SUPER^(); // FB_BA_View
LifeSafety(); // FB_BA_EvtCategory
SafetyMsg(); // FB_BA_EvtCategory
AlarmMsg(); // FB_BA_EvtCategory
FaultMsg(); // FB_BA_EvtCategory
MaintenanceMsg01(); // FB_BA_EvtCategory
MaintenanceMsg02(); // FB_BA_EvtCategory
SystemMsg(); // FB_BA_EvtCategory
ManualOp(); // FB_BA_EvtCategory
OtherMsg(); // FB_BA_EvtCategory

METHOD FB_init : BOOL
VAR_INPUT
	bInitRetains : BOOL; // if TRUE, the retain variables are initialized (warm start / cold start)
	bInCopyCode : BOOL;  // if TRUE, the instance afterwards gets moved into the copy code (online change)
END_VAR
//===================================================================
// Ereigniskategorie - Gefahr für Leben // Event category - Danger to life
// Brandalarm, Überfall // Fire alarm, robbery
LifeSafety.iParent							:= THIS^;
LifeSafety.iLabel							:= LblCtl_EvtCategoryLifeSafty;
LifeSafety.eDPADMode						:= E_BA_DPADMode.eInclude;																						
LifeSafety.EC.nInstanceID						:= EC_ID.NC10;
LifeSafety.EC.iLabel							:= LblFun_ObjectNotificationClass;
LifeSafety.EC.sObjectName						:='{Idx=10}';
LifeSafety.EC.eAlarmMode						:= E_BA_AlarmMode.UserDefined;
LifeSafety.EC.eEventType						:= E_BA_EventType.eAlarm;
LifeSafety.EC.aPriority[1]						:= 10;
LifeSafety.EC.aPriority[2]						:= 11;
LifeSafety.EC.aPriority[3]						:= 12;
LifeSafety.EC.aAcknowledgeRequired[1]			:= TRUE;
LifeSafety.EC.aAcknowledgeRequired[2]			:= FALSE;
LifeSafety.EC.aAcknowledgeRequired[3]			:= TRUE;
//===================================================================		
// Ereigniskategorie - Gefahrenmeldung, Sicherheitsmeldung // Event category - hazard alert, safety message
// Einbruch, unberechtigter Zutritt // Burglary, unauthorised entry
SafetyMsg.iParent							:= THIS^;
SafetyMsg.iLabel							:= LblCtl_EvtCategorySaftyMessage;
SafetyMsg.eDPADMode							:= E_BA_DPADMode.eInclude;																						
SafetyMsg.EC.nInstanceID						:= EC_ID.NC20;
SafetyMsg.EC.iLabel								:= LblFun_ObjectNotificationClass;
SafetyMsg.EC.sObjectName						:='{Idx=20}';
SafetyMsg.EC.eAlarmMode							:= E_BA_AlarmMode.UserDefined;
SafetyMsg.EC.eEventType							:= E_BA_EventType.eAlarm;
SafetyMsg.EC.aPriority[1]						:= 40;
SafetyMsg.EC.aPriority[2]						:= 41;
SafetyMsg.EC.aPriority[3]						:= 42;
SafetyMsg.EC.aAcknowledgeRequired[1]			:= TRUE;
SafetyMsg.EC.aAcknowledgeRequired[2]			:= FALSE;
SafetyMsg.EC.aAcknowledgeRequired[3]			:= TRUE;
//===================================================================//
// Ereigniskategorie - Alarmeldung - Meldung signalisiert Anlagenausfall oder erfordert sofortigen Eingriff 
// Event category - Alarm message - Message signals system failure or requires immediate intervention 
// Sicherheitstemperaturbegrenzer (STB), Sicherheitsdruckbegrenzer (SDB), Übertemperatur der Warmwasserbereitung (WWB), Sicherheitsventile, Hauptpumpen, Keilriemenwächter, Frequenzumformer, Kälteanlagen, Spannungsausfall usw
// Safety temperature limiter, safety pressure limiter, excess temperature of water heating, safety valves, main pumps, V-belt monitors, frequency converters, refrigeration systems, voltage failure, etc.
AlarmMsg.iParent							:= THIS^;
AlarmMsg.iLabel								:= LblCtl_EvtCategoryAlarmMessage;
AlarmMsg.eDPADMode							:= E_BA_DPADMode.eInclude;																						
AlarmMsg.EC.nInstanceID							:= EC_ID.NC30;
AlarmMsg.EC.iLabel								:= LblFun_ObjectNotificationClass;
AlarmMsg.EC.sObjectName							:= '{Idx=30}'	;
AlarmMsg.EC.eAlarmMode							:= E_BA_AlarmMode.UserDefined;
AlarmMsg.EC.eEventType							:= E_BA_EventType.eAlarm;
AlarmMsg.EC.aPriority[1]						:= 70;
AlarmMsg.EC.aPriority[2]						:= 71;
AlarmMsg.EC.aPriority[3]						:= 72;
AlarmMsg.EC.aAcknowledgeRequired[1]				:= TRUE;
AlarmMsg.EC.aAcknowledgeRequired[2]				:= FALSE;
AlarmMsg.EC.aAcknowledgeRequired[3]				:= TRUE;

//===================================================================
// Ereigniskategorie - Störungsmeldung - Meldung weist auf einen anormalen Betriebszustand hin
// Event category - malfunction message - message indicates abnormal operating condition
// Temperaturwächter (TW), Druckwächter (DW), Temperaturüberwachung von Wärmetauscher (WT) und WWB, Motorschutz, Aufzug-Sammelstörmeldung, Netzdrücke usw.
// Temperature monitor, pressure monitor, temperature monitoring of heat exchanger and water heating, motor protection, lift collective fault signal, mains pressures, etc.
FaultMsg.iParent							:= THIS^;
FaultMsg.iLabel								:= LblCtl_EvtCategoryFaultMessage;
FaultMsg.eDPADMode							:= E_BA_DPADMode.eInclude;																						
FaultMsg.EC.nInstanceID							:= EC_ID.NC40;
FaultMsg.EC.iLabel								:= LblFun_ObjectNotificationClass;
FaultMsg.EC.sObjectName							:= '{Idx=40}'	;
FaultMsg.EC.eAlarmMode							:= E_BA_AlarmMode.UserDefined;
FaultMsg.EC.eEventType							:= E_BA_EventType.eDisturb;
FaultMsg.EC.aPriority[1]						:= 100;
FaultMsg.EC.aPriority[2]						:= 101;
FaultMsg.EC.aPriority[3]						:= 102;
FaultMsg.EC.aAcknowledgeRequired[1]				:= TRUE;
FaultMsg.EC.aAcknowledgeRequired[2]				:= FALSE;
FaultMsg.EC.aAcknowledgeRequired[3]				:= FALSE;
//===================================================================
// Ereigniskategorie - Wartungsmeldung, Hinweis auf Wartungsaktivität o.ä.
// Event category - Maintenance message Maintenance message, indication of maintenance activity or similar.
// Betriebsstunden, Behälterstand, Reparaturschalter usw.
// Operating hours, tank level, repair switch, etc.
MaintenanceMsg01.iParent					:= THIS^;
MaintenanceMsg01.iLabel						:= LblCtl_EvtCategoryMaintenanceMessage;
MaintenanceMsg01.eDPADMode					:= E_BA_DPADMode.eInclude;																						
MaintenanceMsg01.EC.nInstanceID					:= EC_ID.NC50;
MaintenanceMsg01.EC.iLabel						:= LblFun_ObjectNotificationClass;
MaintenanceMsg01.EC.sObjectName					:= '{Idx=50}'	;
MaintenanceMsg01.EC.eAlarmMode					:= E_BA_AlarmMode.UserDefined;
MaintenanceMsg01.EC.eEventType					:= E_BA_EventType.eMaintenance;
MaintenanceMsg01.EC.aPriority[1]				:= 130;
MaintenanceMsg01.EC.aPriority[2]				:= 131;
MaintenanceMsg01.EC.aPriority[3]				:= 132;
MaintenanceMsg01.EC.aAcknowledgeRequired[1]		:= TRUE;
MaintenanceMsg01.EC.aAcknowledgeRequired[2]		:= FALSE;
MaintenanceMsg01.EC.aAcknowledgeRequired[3]		:= FALSE;

// Filterende erreicht, Filter verschmutzt usw.
// Filter end reached, filter dirty, etc.
MaintenanceMsg02.iParent					:= THIS^;
MaintenanceMsg02.iLabel						:= LblCtl_EvtCategoryMaintenanceMessage;
MaintenanceMsg02.eDPADMode					:= E_BA_DPADMode.eInclude;																						
MaintenanceMsg02.EC.nInstanceID					:= EC_ID.NC51;
MaintenanceMsg02.EC.iLabel						:= LblFun_ObjectNotificationClass;
MaintenanceMsg02.EC.sObjectName					:= '{Idx=51}'	;
MaintenanceMsg02.EC.eAlarmMode					:= E_BA_AlarmMode.UserDefined;
MaintenanceMsg02.EC.eEventType					:= E_BA_EventType.eMaintenance;
MaintenanceMsg02.EC.aPriority[1]				:= 135;
MaintenanceMsg02.EC.aPriority[2]				:= 136;
MaintenanceMsg02.EC.aPriority[3]				:= 137;
MaintenanceMsg02.EC.aAcknowledgeRequired[1]		:= TRUE;
MaintenanceMsg02.EC.aAcknowledgeRequired[2]		:= FALSE;
MaintenanceMsg02.EC.aAcknowledgeRequired[3]		:= FALSE;
//===================================================================
//===================================================================
// Ereigniskategorie - Systemmeldung, Störungsmeldung aus GA-System
// Event category - System message, System message, Fault message from building automation system
// Gerätestörung, Batteriemeldung, Kommunikationsunterbrechung usw.
// Unit malfunction, battery message, communication interruption, etc.
SystemMsg.iParent							:= THIS^;
SystemMsg.iLabel							:= LblCtl_EvtCategorySystem;
SystemMsg.eDPADMode							:= E_BA_DPADMode.eInclude;																						
SystemMsg.EC.nInstanceID						:= EC_ID.NC60;
SystemMsg.EC.iLabel								:= LblFun_ObjectNotificationClass;
SystemMsg.EC.sObjectName						:='{Idx=60}';
SystemMsg.EC.eAlarmMode							:= E_BA_AlarmMode.UserDefined;
SystemMsg.EC.eEventType							:= E_BA_EventType.eNotification;
SystemMsg.EC.aPriority[1]						:= 180;
SystemMsg.EC.aPriority[2]						:= 181;
SystemMsg.EC.aPriority[3]						:= 182;
SystemMsg.EC.aAcknowledgeRequired[1]			:= FALSE;
SystemMsg.EC.aAcknowledgeRequired[2]			:= FALSE;
SystemMsg.EC.aAcknowledgeRequired[3]			:= FALSE;
//===================================================================//
//	Ereigniskategorie - Manual operation, Handeingriff
ManualOp.iParent							:= THIS^;
ManualOp.iLabel								:= LblCtl_EvtCategoryManualOperation;
ManualOp.eDPADMode							:= E_BA_DPADMode.eInclude;																						
ManualOp.EC.nInstanceID							:= EC_ID.NC70;
ManualOp.EC.iLabel								:= LblFun_ObjectNotificationClass;
ManualOp.EC.sObjectName							:='{Idx=70}';
ManualOp.EC.eAlarmMode							:= E_BA_AlarmMode.UserDefined;
ManualOp.EC.eEventType							:= E_BA_EventType.eOther;
ManualOp.EC.aPriority[1]						:= 220;
ManualOp.EC.aPriority[2]						:= 220;
ManualOp.EC.aPriority[3]						:= 220;
ManualOp.EC.aAcknowledgeRequired[1]				:= FALSE;
ManualOp.EC.aAcknowledgeRequired[2]				:= FALSE;
ManualOp.EC.aAcknowledgeRequired[3]				:= FALSE;
//===================================================================//
// Ereigniskategorie - Freibleibend, Sonstige Meldungen
// Event category - Other message, Not binding, Other messages
// Betriebszustandswechsel, Betriebsarten, Trendspeicher voll usw.
// Operating status change, operating modes, trend memory full, etc.
OtherMsg.iParent							:= THIS^;
OtherMsg.iLabel								:= LblCtl_EvtCategoryOther;
OtherMsg.eDPADMode							:= E_BA_DPADMode.eInclude;																						
OtherMsg.EC.nInstanceID							:= EC_ID.NC80;
OtherMsg.EC.iLabel								:= LblFun_ObjectNotificationClass;
OtherMsg.EC.sObjectName							:='{Idx=80}';
OtherMsg.EC.eAlarmMode							:= E_BA_AlarmMode.UserDefined;
OtherMsg.EC.eEventType							:= E_BA_EventType.eOther;
OtherMsg.EC.aPriority[1]						:= 230;
OtherMsg.EC.aPriority[2]						:= 231;
OtherMsg.EC.aPriority[3]						:= 232;
OtherMsg.EC.aAcknowledgeRequired[1]				:= FALSE;
OtherMsg.EC.aAcknowledgeRequired[2]				:= FALSE;
OtherMsg.EC.aAcknowledgeRequired[3]				:= FALSE;
END_METHOD

END_FUNCTION_BLOCK

// ---- Templates/POUs/Trade/BuildingAutomation/Communication/FB_BA_AdsComClient.TcPOU
FUNCTION_BLOCK FB_BA_AdsComClient EXTENDS FB_BA_VIEW
VAR_INPUT
END_VAR
VAR_OUTPUT
END_VAR
VAR_INPUT CONSTANT
	WeatherStation					: FB_BA_RawSubscriber;
	WeatherStationError				: FB_BA_BV;											

	GeneralSettings					: FB_BA_RawSubscriber;												
	GeneralSettingsError			: FB_BA_BV;			
END_VAR
VAR
END_VAR

// Error-notification
WeatherStationError(bEnPgm := TRUE, bValPgm := WeatherStation.bError); // FB_BA_BV
GeneralSettingsError(bEnPgm := TRUE, bValPgm := GeneralSettings.bError); // FB_BA_BV
// variable, on which the error-notification is written
Site.bWeatherStation_Error := WeatherStationError.bEvent;
// variable, on which the subscribed data is written
// because this variable is an announcement for the suscriber,
// where to write the data, it is declared as an input
// error-delay: see FB_Init
WeatherStation(xData := Site.stWeatherStation); // FB_BA_RawSubscriber
Site.bGeneralSettings_Error := GeneralSettingsError.bEvent;
GeneralSettings(xData := Site.stGeneralSettings); // FB_BA_RawSubscriber
SUPER^(); // FB_BA_VIEW

METHOD FB_init : BOOL
VAR_INPUT
	bInitRetains : BOOL; // if TRUE, the retain variables are initialized (warm start / cold start)
	bInCopyCode : BOOL;  // if TRUE, the instance afterwards gets moved into the copy code (online change)
END_VAR
WeatherStation.Subject							:= Site.WeatherStation_Subject;		// instance-name of the publisher in the source
WeatherStation.sTarget							:= Site.WeatherStation_NetId;		// AMS-Net-Id of the publishing controller
WeatherStation.tReadInterval					:= T#5S;							// subscribe-interval
WeatherStation.tReadTolerance					:= T#60S;							// delay time, until an erroneous communication will be displayed at the error-output of the subscriber

WeatherStationError.iParent						:= THIS^;
WeatherStationError.iLabel						:= LblAgg_WeatherStationComm;
WeatherStationError.sActiveText 				:= txtEvent_Triggered;
WeatherStationError.sInactiveText 				:= txtEvent_Normal;
WeatherStationError.bEnManualRm					:= FALSE;	//	Priority  8	
WeatherStationError.bValManualRm				:= FALSE;	//	Priority  8
WeatherStationError.nEventClassID				:= EC_ID.NC30;
WeatherStationError.stTimeDelay.nToNormal		:= 0;
WeatherStationError.stTimeDelay.nToAbnormal		:= 0;
WeatherStationError.bAlarmValue					:= TRUE;
WeatherStationError.aEventTransitionText[1]		:= txtEvent_Disturb;
WeatherStationError.aEventTransitionText[2]		:= txtEvent_None;
WeatherStationError.aEventTransitionText[3]		:= txtEvent_Normal;
WeatherStationError.bEventDetectionEnable		:= TRUE;
WeatherStationError.eEnPlantLock				:= E_BA_LockPriority.eNoLock;

GeneralSettings.Subject							:= Site.GeneralSettings_Subject;	// instance-name of the publisher in the source
GeneralSettings.sTarget							:= Site.GeneralSettings_NetId;		// AMS-Net-Id of the publishing controller
GeneralSettings.tReadInterval					:= T#5S;							// subscribe-interval
GeneralSettings.tReadTolerance					:= T#60S;							// delay time, until an erroneous communication will be displayed at the error-output of the subscriber

GeneralSettingsError.iParent					:= THIS^;
GeneralSettingsError.iLabel						:= LblAgg_GeneralSettingsCom;
//GeneralSettingsError.sObjectName				:= F_BA_CONCAT06(s01:= Seperator.sAgg_ObjName, s02:= Agg_GeneralSettingsCom_ObjName, s03:= '02', s04:= Seperator.sFun_ObjName, s05:= Fun_Fault_ObjName, s06:= '01');  
//GeneralSettingsError.sDescription				:= F_BA_CONCAT06(s01:= Seperator.sAgg_Descr, s02:= Agg_GeneralSettingsCom_Descr, s03:= '', s04:= Seperator.sFun_Descr, s05:= Fun_Fault_Descr, s06:= ''); 	
GeneralSettingsError.sActiveText 				:= txtEvent_Triggered;
GeneralSettingsError.sInactiveText 				:= txtEvent_Normal;
GeneralSettingsError.bEnManualRm				:= FALSE;	//	Priority  8	
GeneralSettingsError.bValManualRm				:= FALSE;	//	Priority  8
GeneralSettingsError.nEventClassID				:= EC_ID.NC30;
GeneralSettingsError.stTimeDelay.nToNormal		:= 0;
GeneralSettingsError.stTimeDelay.nToAbnormal	:= 0;
GeneralSettingsError.bAlarmValue				:= TRUE;
GeneralSettingsError.aEventTransitionText[1]	:= txtEvent_Disturb;
GeneralSettingsError.aEventTransitionText[2]	:= txtEvent_None;
GeneralSettingsError.aEventTransitionText[3]	:= txtEvent_Normal;
GeneralSettingsError.bEventDetectionEnable		:= TRUE;
GeneralSettingsError.eEnPlantLock				:= E_BA_LockPriority.eNoLock;
END_METHOD

END_FUNCTION_BLOCK

// ---- Templates/POUs/Trade/HeatingSystem/General/FB_BA_HtgLmt.TcPOU
{region '#Template'}
	{attribute 'Version' := '5.0.0.0'}
	{attribute 'Tags' := '"LCID": "1031", "Text": "H, General, HtgCir, Operating mode"'}
	{attribute 'Tags' := '"LCID": "1033", "Text": "H, General, HtgCir, Operating mode"'}
	{attribute 'Using' := '"Type": "Template", "URI": "BA2_Param"'}
	{attribute 'Description' := '"LCID": "1031", "Text": "Heizgrenzwert"'}
	{attribute 'Description' := '"LCID": "1033", "Text": "Heating limit"'}
{endregion}
FUNCTION_BLOCK FB_BA_HtgLmt EXTENDS FB_BA_View
VAR_INPUT
	fIn						: REAL;
END_VAR
VAR_OUTPUT
	bQ						: BOOL;
END_VAR
VAR_INPUT CONSTANT
	Sp						: FB_BA_AV_Op;	
	Q						: FB_BA_BV_Op;		
END_VAR	
VAR
	Swi2P					: FB_BA_Swi2P;
END_VAR
VAR // added by the converter: edge detectors and wires of the graphical bodies
    _w1 : ANY;
END_VAR

SUPER^(); // FB_BA_View
Sp(); // FB_BA_AV_Op
_w1 := LIMIT(10, Sp.fPresentValue, 32);
Swi2P(bEn := TRUE, fIn := fIn, fOn := _w1, fOff := _w1 + 0.5); // FB_BA_Swi2P
Q(bValuePgm := Swi2P.bQ); // FB_BA_BV_Op
bQ := Q.bPresentValue;

METHOD FB_init : BOOL
VAR_INPUT
	bInitRetains : BOOL; // if TRUE, the retain variables are initialized (warm start / cold start)
	bInCopyCode : BOOL;  // if TRUE, the instance afterwards gets moved into the copy code (online change)
END_VAR
Sp.iParent			:= THIS^;
Sp.iLabel			:= LblFun_Setpoint; 
Sp.eUnit			:= E_BA_Unit.eTemperature_DegreesCelsius;  
Sp.fValueRm			:= 16.0;
Sp.fCOVIncrement	:= BA2_Param.fDefCOVIncrement;							

Q.iParent			:= THIS^;
Q.iLabel			:= LblFun_OperationalMessage; 
Q.sActiveText		:= txtEvent_On;
Q.sInactiveText		:= txtEvent_Off;
Q.bValueRm			:= FALSE;								
Q.eToggleMode 		:= E_BA_ToggleMode.eSwitch;
END_METHOD

END_FUNCTION_BLOCK

// ---- Templates/POUs/Trade/HeatingSystem/Setpoint/FB_BA_H_HtgCir_Sp.TcPOU
{region '#Template'}
	{attribute 'Version' := '5.0.0.0'}
	{attribute 'Tags' := '"LCID": "1031", "Text": "H, Heating circuit, HtgCir, Setpoint"'}
	{attribute 'Tags' := '"LCID": "1033", "Text": "H, Heating circuit, HtgCir, Setpoint"'}
	{attribute 'Using' := '"Type": "Template", "URI": "BA2_Param"'}
	{attribute 'Using' := '"Type": "Template", "URI": "E_BA_EnergyLvl"'}		 
	{attribute 'Description' := '"LCID": "1031", "Text": "Sollwert Heizkreis"'}
	{attribute 'Description' := '"LCID": "1033", "Text": "Setpoint heating circuit"'}
{endregion}
FUNCTION_BLOCK FB_BA_H_HtgCir_Sp EXTENDS FB_BA_View
VAR_INPUT
	eOpMod					: E_BA_EnergyLvl;
	fSpFrstProtec			: REAL;
	fTWthDamp				: REAL;
END_VAR
VAR_OUTPUT
	fSpFlWT							: REAL;
END_VAR
VAR_INPUT CONSTANT
	NgtOffs					: FB_BA_AV_Op;	
	SpFlWT					: FB_BA_AV_Op;		
	HtgCrv					: FB_BA_Scale_04; 
END_VAR
VAR
	PrioSwi					: FB_BA_MMUX_R04;
END_VAR

// note: 1 stored wires end on pins the file does not list and are not shown
SUPER^(); // FB_BA_View
NgtOffs(); // FB_BA_AV_Op
HtgCrv(fX := fTWthDamp); // FB_BA_Scale_04
PrioSwi(
    bEn := TRUE,
    nSel := eOpMod,
    nEn01 := E_BA_EnergyLvl.eComfort,
    fVal01 := HtgCrv.fY,
    nEn02 := E_BA_EnergyLvl.eEconomy,
    fVal02 := HtgCrv.fY - ABS(NgtOffs.fPresentValue),
    nEn03 := E_BA_EnergyLvl.eProtection,
    fVal03 := fSpFrstProtec); // FB_BA_MMUX_R04
SpFlWT(fValuePgm := PrioSwi.fVal); // FB_BA_AV_Op
fSpFlWT := SpFlWT.fPresentValue;

METHOD FB_init : BOOL
VAR_INPUT
	bInitRetains : BOOL; // if TRUE, the retain variables are initialized (warm start / cold start)
	bInCopyCode : BOOL;  // if TRUE, the instance afterwards gets moved into the copy code (online change)
END_VAR
NgtOffs.iParent				:= THIS^;
NgtOffs.iLabel				:= LblCtl_OffsetNightSetpoint; 
NgtOffs.eUnit				:= E_BA_Unit.eTemperature_DegreesCelsius;  
NgtOffs.fValueRm			:= 8.0;
NgtOffs.fCOVIncrement		:= BA2_Param.fDefCOVIncrement;							

SpFlWT.iParent				:= THIS^;
SpFlWT.iLabel				:= LblFun_Setpoint; 
SpFlWT.eUnit				:= E_BA_Unit.eTemperature_DegreesCelsius;  
SpFlWT.fCOVIncrement		:= BA2_Param.fDefCOVIncrement;							

HtgCrv.iParent				:= THIS^;										
HtgCrv.iLabel				:= LblCtl_HeatingCurve; 
HtgCrv.eDPADMode			:= E_BA_DPADMode.eIncludeDescription; 
HtgCrv.X1.fValueRm			:= 15.0;
HtgCrv.X2.fValueRm			:= 0.0;
HtgCrv.X3.fValueRm			:= -10.0;
HtgCrv.X4.fValueRm			:= -20.0;
HtgCrv.Y1.fValueRm			:= 25.0;
HtgCrv.Y2.fValueRm			:= 40.0;
HtgCrv.Y3.fValueRm			:= 55.0;
HtgCrv.Y4.fValueRm			:= 65.0;
HtgCrv.YMin.fValueRm		:= 5.0;
HtgCrv.YMax.fValueRm		:= 80.0;
END_METHOD

END_FUNCTION_BLOCK

// ---- Templates/POUs/Universal/Control/Scale/FB_BA_Scale_04.TcPOU
{region '#Template'}
	{attribute 'Version' := '5.0.0.0'}
	{attribute 'Tags' := '"LCID": "1031", "Text": "Universal, Control, Scaling"'}
	{attribute 'Tags' := '"LCID": "1033", "Text": "Universal, Control, Scaling"'}
	{attribute 'Using' := '"Type": "Template", "URI": "BA2_Param"'}
	{attribute 'Description' := '"LCID": "1031", "Text": "Skalierung"'}
	{attribute 'Description' := '"LCID": "1033", "Text": "Scaling"'}
{endregion}
FUNCTION_BLOCK FB_BA_Scale_04 EXTENDS FB_BA_View
VAR_INPUT
	fX			: REAL;
END_VAR
VAR_OUTPUT
	fY			: REAL;
END_VAR
VAR_INPUT CONSTANT
	X1			: FB_BA_AV_Op;	
	X2			: FB_BA_AV_Op;	
	X3			: FB_BA_AV_Op;	
	X4			: FB_BA_AV_Op;	
	Y1			: FB_BA_AV_Op;	
	Y2			: FB_BA_AV_Op;
	Y3			: FB_BA_AV_Op;
	Y4			: FB_BA_AV_Op;
	YMin		: FB_BA_AV_Op;			
	YMax		: FB_BA_AV_Op;			
	Y			: FB_BA_AV_Op;		
END_VAR
VAR		
	Scale		: FB_BA_Chrct04;
END_VAR

SUPER^(); // FB_BA_View
X1(); // FB_BA_AV_Op
X2(); // FB_BA_AV_Op
X3(); // FB_BA_AV_Op
X4(); // FB_BA_AV_Op
Y1(); // FB_BA_AV_Op
Y2(); // FB_BA_AV_Op
Y3(); // FB_BA_AV_Op
Y4(); // FB_BA_AV_Op
Ymin(); // FB_BA_AV_Op
YMax(); // FB_BA_AV_Op
Scale(
    fX := fX,
    fX01 := X1.fPresentValue,
    fX02 := X2.fPresentValue,
    fX03 := X3.fPresentValue,
    fX04 := X4.fPresentValue,
    fY01 := Y1.fPresentValue,
    fY02 := Y2.fPresentValue,
    fY03 := Y3.fPresentValue,
    fY04 := Y4.fPresentValue,
    fYMin := Ymin.fPresentValue,
    fYMax := YMax.fPresentValue); // FB_BA_Chrct04
Y(fValuePgm := Scale.fCalcVal); // FB_BA_AV_Op
fY := Y.fPresentValue;

METHOD FB_init : BOOL
VAR_INPUT
	bInitRetains : BOOL; // if TRUE, the retain variables are initialized (warm start / cold start)
	bInCopyCode : BOOL;  // if TRUE, the instance afterwards gets moved into the copy code (online change)
END_VAR
X1.iParent			:= THIS^;
X1.iLabel		:= LblCtl_X01;  							 	 
X1.eUnit			:= E_BA_Unit.eTemperature_DegreesCelsius;						 	 
X1.fValueRm			:= 15.0;
X1.fCOVIncrement	:= BA2_Param.fDefCOVIncrement;		

X2.iParent			:= THIS^;
X2.iLabel		:= LblCtl_X02;  								 	 
X2.eUnit			:= E_BA_Unit.eTemperature_DegreesCelsius;						 	 
X2.fValueRm			:= 0.0;
X2.fCOVIncrement	:= BA2_Param.fDefCOVIncrement;		

X3.iParent			:= THIS^;
X3.iLabel		:= LblCtl_X03;  								 	 
X3.eUnit			:= E_BA_Unit.eTemperature_DegreesCelsius;						 	 
X3.fValueRm			:= -20.0;
X3.fCOVIncrement	:= BA2_Param.fDefCOVIncrement;			

X4.iParent			:= THIS^;
X4.iLabel		:= LblCtl_X04;  									 	 
X4.eUnit			:= E_BA_Unit.eTemperature_DegreesCelsius;						 	 
X4.fValueRm			:= -20.0;
X4.fCOVIncrement	:= BA2_Param.fDefCOVIncrement;		

Y1.iParent			:= THIS^;
Y1.iLabel		:= LblCtl_Y01;  			 	 
Y1.eUnit			:= E_BA_Unit.eTemperature_DegreesCelsius;						 	 
Y1.fValueRm			:= 25.0;
Y1.fCOVIncrement	:= BA2_Param.fDefCOVIncrement;		

Y2.iParent			:= THIS^;
Y2.iLabel		:= LblCtl_Y02;  							 	 
Y2.eUnit			:= E_BA_Unit.eTemperature_DegreesCelsius;						 	 
Y2.fValueRm			:= 40.0;
Y2.fCOVIncrement	:= BA2_Param.fDefCOVIncrement;		

Y3.iParent			:= THIS^;
Y3.iLabel			:= LblCtl_Y03;  							 	 
Y3.eUnit			:= E_BA_Unit.eTemperature_DegreesCelsius;						 	 
Y3.fValueRm			:= 60.0;
Y3.fCOVIncrement	:= BA2_Param.fDefCOVIncrement;		


Y4.iParent			:= THIS^;
Y4.iLabel			:= LblCtl_Y04;  									 	 
Y4.eUnit			:= E_BA_Unit.eTemperature_DegreesCelsius;						 	 
Y4.fValueRm			:= 65.0;
Y4.fCOVIncrement	:= BA2_Param.fDefCOVIncrement;		

YMin.iParent		:= THIS^;
YMin.iLabel			:= LblFun_MinimumValue;										 	 
YMin.eUnit			:= E_BA_Unit.eTemperature_DegreesCelsius;						 	 
YMin.fValueRm		:= 5.0;
YMin.fCOVIncrement	:= BA2_Param.fDefCOVIncrement;		

YMax.iParent		:= THIS^;
YMax.iLabel			:= LblFun_MaximumValue;							 	 
YMax.eUnit			:= E_BA_Unit.eTemperature_DegreesCelsius;						 	 
YMax.fValueRm		:= 80.0;
YMax.fCOVIncrement	:= BA2_Param.fDefCOVIncrement;		

Y.iParent			:= THIS^;
Y.iLabel			:= LblFun_SetpointCalculated;										 	 
Y.eUnit				:= E_BA_Unit.eTemperature_DegreesCelsius;	
Y.fCOVIncrement		:= BA2_Param.fDefCOVIncrement;
END_METHOD

END_FUNCTION_BLOCK

// ---- Templates/POUs/Universal/Aggregat/Analog/FB_BA_ActuatorAV.TcPOU
{region '#Template'}
	{attribute 'Version' := '5.0.0.0'}
	{attribute 'Tags' := '"LCID": "1031", "Text": "Universal, Analog, Aggregate"'}
	{attribute 'Tags' := '"LCID": "1033", "Text": "Universal, Analog, Aggregate"'}
	{attribute 'Using' := '"Type": "Template", "URI": "EC_ID"'}
	{attribute 'Using' := '"Type": "Template", "URI": "BA2_Param"'}
	{attribute 'Description' := '"LCID": "1031", "Text": "AV"'}
	{attribute 'Description' := '"LCID": "1033", "Text": "AV"'}
{endregion}
FUNCTION_BLOCK FB_BA_ActuatorAV EXTENDS FB_BA_View
VAR_INPUT
	stCmd					: ST_BA_Analog;	
END_VAR
VAR_OUTPUT
	fPresentValue		: REAL;
	bDst				: BOOL;
	eActivePrio			: E_BA_Priority;	
END_VAR
VAR_INPUT CONSTANT
	Val					: FB_BA_AV;		
	PlantLock			: FB_BA_PlantLock;	
END_VAR
VAR
	bPrioSfty				: BOOL;
	bPrioCrit				: BOOL;	
END_VAR

SUPER^(); // FB_BA_View
PlantLock(); // FB_BA_PlantLock
bPrioSfty := PlantLock.bPrioHigh OR PlantLock.bPrioLocalHigh;
bPrioCrit := PlantLock.bPrioMedium OR PlantLock.bPrioLocalMedium;
bDst := bPrioSfty OR bPrioCrit;
Val(
    bEnSfty := stCmd.bEnSfty OR bPrioSfty,
    fValSfty := SEL(bPrioSfty, stCmd.fValSfty, 0),
    bEnCrit := stCmd.bEnCrit OR bPrioCrit,
    fValCrit := SEL(bPrioCrit, stCmd.fValCrit, 0),
    bEnPgm := stCmd.bEnPgm,
    fValPgm := stCmd.fValPgm); // FB_BA_AV
fPresentValue := Val.fPresentValue;
eActivePrio := Val.eActivePrio;

METHOD FB_init : BOOL
VAR_INPUT
	bInitRetains : BOOL; // if TRUE, the retain variables are initialized (warm start / cold start)
	bInCopyCode : BOOL;  // if TRUE, the instance afterwards gets moved into the copy code (online change)
END_VAR
PlantLock.Parent				:= THIS^;		

Val.iParent						:= THIS^;
Val.iLabel						:= LblFun_ControlSignal;  
Val.eUnit						:= E_BA_Unit.eOther_Percent;
Val.fCOVIncrement				:= BA2_Param.fDefCOVIncrement;
Val.bEnManualRm					:= FALSE;	//	Priority  8	
Val.fValManualRm				:= 0.0;		//	Priority  8
Val.fDefaultValue				:= 0.0;	
Val.nEventClassID				:= EC_ID.NC80;
Val.stTimeDelay.nToNormal		:= BA2_Param.nDefTimeDelay_ToNormal;
Val.stTimeDelay.nToAbnormal		:= BA2_Param.nDefTimeDelay_ToAbnormal;
Val.stHighLimit.bEnable			:= FALSE;
Val.stHighLimit.fValue			:= 0.0;		
Val.stLowLimit.bEnable			:= FALSE;
Val.stLowLimit.fValue			:= 0.0;
Val.fLimitDeadband 				:= BA2_Param.fDefLimitDeadband;
Val.bAcknowledgeRm				:= FALSE;	
Val.aEventTransitionText[1]		:= txtEvent_Disturb;
Val.aEventTransitionText[2]		:= txtEvent_None;
Val.aEventTransitionText[3]		:= txtEvent_Normal;
Val.bEventDetectionEnable		:= FALSE;
Val.eEnPlantLock				:= E_BA_LockPriority.eNoLock;
END_METHOD

END_FUNCTION_BLOCK

// ---- Templates/POUs/Universal/Aggregat/Modulation/FB_BA_ActuatorMdlt.TcPOU
{region '#Template'}
	{attribute 'Version' := '5.0.0.0'}
	{attribute 'Tags' := '"LCID": "1031", "Text": "Universal, Analog, Aggregate"'}
	{attribute 'Tags' := '"LCID": "1033", "Text": "Universal, Analog, Aggregate"'}
	{attribute 'Using' := '"Type": "Template", "URI": "EC_ID"'}
	{attribute 'Using' := '"Type": "Template", "URI": "BA2_Param"'}
	{attribute 'Description' := '"LCID": "1031", "Text": "Aktor analog"'}
	{attribute 'Description' := '"LCID": "1033", "Text": "Actuator analog"'}
{endregion}
FUNCTION_BLOCK FB_BA_ActuatorMdlt EXTENDS FB_BA_View
VAR_INPUT
	stCmd					: ST_BA_Mdlt;	
	fValPgm					: REAL;
END_VAR
VAR_OUTPUT
	fMdlt					: REAL;
	bDst					: BOOL;
	eActivePrio				: E_BA_Priority;
END_VAR
VAR_INPUT CONSTANT PERSISTENT
	{attribute 'parameterCategory' := 'Behaviour'}
	fMinModulation 				: REAL := 20;
	{attribute 'parameterCategory' := 'Behaviour'}
	fMaxModulation 				: REAL := 100;
END_VAR
VAR_INPUT CONSTANT
	Mdlt					: FB_BA_AO_Raw;
	PlantLock				: FB_BA_PlantLock;	
END_VAR
VAR
	bPrioSfty					: BOOL;
	bPrioCrit					: BOOL;	
	
	PrioSwiVal					: FB_BA_PrioSwi_UDI04;	
	MuxMdlt						: FB_BA_MMUX_R04;
END_VAR

SUPER^(); // FB_BA_View
PlantLock(); // FB_BA_PlantLock
bPrioSfty := PlantLock.bPrioHigh OR PlantLock.bPrioLocalHigh;
bPrioCrit := PlantLock.bPrioMedium OR PlantLock.bPrioLocalMedium;
bDst := bPrioSfty OR bPrioCrit;
PrioSwiVal(
    bEn01 := stCmd.bEnSfty,
    nVal01 := stCmd.eValSfty,
    bEn02 := stCmd.bEnCrit,
    nVal02 := stCmd.eValCrit,
    bEn03 := stCmd.bEnPgm,
    nVal03 := stCmd.eValPgm); // FB_BA_PrioSwi_UDI04
MuxMdlt(
    bEn := TRUE,
    nSel := PrioSwiVal.nVal,
    nEn01 := E_BA_Mdlt.eOff,
    fVal01 := 0,
    nEn02 := E_BA_Mdlt.eOn,
    fVal02 := fValPgm,
    nEn03 := E_BA_Mdlt.eMin,
    fVal03 := fMinModulation,
    nEn04 := E_BA_Mdlt.eMax,
    fVal04 := fMaxModulation); // FB_BA_MMUX_R04
Mdlt(
    bEnSfty := stCmd.bEnSfty,
    fValSfty := SEL(bPrioSfty, MuxMdlt.fVal, 0),
    bEnCrit := stCmd.bEnCrit,
    fValCrit := SEL(bPrioCrit, MuxMdlt.fVal, 0),
    bEnPgm := stCmd.bEnPgm,
    fValPgm := MuxMdlt.fVal); // FB_BA_AO_Raw
fMdlt := Mdlt.fPresentValue;
eActivePrio := Mdlt.eActivePrio;

METHOD FB_init : BOOL
VAR_INPUT
	bInitRetains : BOOL; // if TRUE, the retain variables are initialized (warm start / cold start)
	bInCopyCode : BOOL;  // if TRUE, the instance afterwards gets moved into the copy code (online change)
END_VAR
PlantLock.Parent				:= THIS^;		

Mdlt.iParent					:= THIS^;
Mdlt.iLabel						:= LblFun_ControlSignal;
Mdlt.eUnit						:= E_BA_Unit.eOther_Percent;
Mdlt.fResolution 				:= 0.003051851;
Mdlt.fScaleOffset 				:= 0;
Mdlt.fCOVIncrement				:= BA2_Param.fDefCOVIncrement;
Mdlt.bEnManualRm				:= FALSE;	//	Priority  8	
Mdlt.fValManualRm				:= 0.0;		//	Priority  8
Mdlt.nEventClassID				:= EC_ID.NC80;
Mdlt.stTimeDelay.nToNormal		:= BA2_Param.nDefTimeDelay_ToNormal;
Mdlt.stTimeDelay.nToAbnormal	:= BA2_Param.nDefTimeDelay_ToAbnormal;
Mdlt.stHighLimit.bEnable		:= FALSE;
Mdlt.stHighLimit.fValue			:= 0.0;		
Mdlt.stLowLimit.bEnable			:= FALSE;
Mdlt.stLowLimit.fValue			:= 0.0;
Mdlt.fLimitDeadband 			:= BA2_Param.fDefLimitDeadband;
Mdlt.aEventTransitionText[1]	:= txtEvent_Disturb;
Mdlt.aEventTransitionText[2]	:= txtEvent_None;
Mdlt.aEventTransitionText[3]	:= txtEvent_Normal;
Mdlt.bEventDetectionEnable		:= FALSE;
Mdlt.eEnPlantLock				:= E_BA_LockPriority.eNoLock;
END_METHOD

END_FUNCTION_BLOCK

// ---- Templates/POUs/Universal/Aggregat/Multistate/FB_BA_ActuatorMultistate.TcPOU
{region '#Template'}
	{attribute 'Version' := '5.0.0.0'}
	{attribute 'Tags' := '"LCID": "1031", "Text": "Universal, Multistate, Aggregate"'}
	{attribute 'Tags' := '"LCID": "1033", "Text": "Universal, Multistate, Aggregate"'}
	{attribute 'Using' := '"Type": "Template", "URI": "EC_ID"'}
	{attribute 'Using' := '"Type": "Template", "URI": "BA2_Param"'}
	{attribute 'Description' := '"LCID": "1031", "Text": "Aktor multistate"'}
	{attribute 'Description' := '"LCID": "1033", "Text": "Actuator multistate"'}
{endregion}			 
FUNCTION_BLOCK FB_BA_ActuatorMultistate EXTENDS FB_BA_View
VAR_INPUT
	stCmd					: ST_BA_Multistate;	
END_VAR
VAR_OUTPUT
	nCmd					: UDINT;
	bDst					: BOOL;
	eActivePrio				: E_BA_Priority;
END_VAR
VAR_INPUT CONSTANT	
	Cmd						: FB_BA_MO_Raw;	
	PlantLock				: FB_BA_PlantLock;	
END_VAR
VAR
	bPrioSfty				: BOOL;
	bPrioCrit				: BOOL;	
END_VAR
VAR // added by the converter: edge detectors and wires of the graphical bodies
    _w1 : ANY;
END_VAR

SUPER^(); // FB_BA_View
PlantLock(); // FB_BA_PlantLock
bPrioSfty := PlantLock.bPrioHigh OR PlantLock.bPrioLocalHigh;
bPrioCrit := PlantLock.bPrioMedium OR PlantLock.bPrioLocalMedium;
bDst := bPrioSfty OR bPrioCrit;
Cmd(
    bEnSfty := stCmd.bEnSfty OR bPrioSfty,
    nValSfty := SEL(bPrioSfty, stCmd.nValSfty, 1),
    bEnCrit := stCmd.bEnCrit OR bPrioCrit,
    nValCrit := _w1,
    bEnPgm := stCmd.bEnPgm,
    nValPgm := stCmd.nValPgm); // FB_BA_MO_Raw
_w1 := SEL(bPrioCrit, stCmd.nValCrit, 1);
nCmd := Cmd.nPresentValue;
eActivePrio := Cmd.eActivePrio;

METHOD FB_init : BOOL
VAR_INPUT
	bInitRetains : BOOL; // if TRUE, the retain variables are initialized (warm start / cold start)
	bInCopyCode : BOOL;  // if TRUE, the instance afterwards gets moved into the copy code (online change)
END_VAR
PlantLock.Parent				:= THIS^;	

Cmd.iParent						:= THIS^;
Cmd.iLabel						:= LblFun_SwitchingCommand;
Cmd.aStateText[1]				:= txtEvent_Stop;
Cmd.aStateText[2]				:= txtEvent_Open;
Cmd.aStateText[3]				:= txtEvent_Close;
Cmd.bEnManualRm					:= FALSE;	//	Priority  8	
Cmd.nValManualRm				:= 1;		//	Priority  8
Cmd.nDefaultValue				:= 1;	
Cmd.nEventClassID				:= EC_ID.NC80;
Cmd.stTimeDelay.nToNormal		:= BA2_Param.nDefTimeDelay_ToNormal;
Cmd.stTimeDelay.nToAbnormal		:= BA2_Param.nDefTimeDelay_ToAbnormal;
Cmd.aEventTransitionText[1]		:= txtEvent_Disturb;
Cmd.aEventTransitionText[2]		:= txtEvent_None;
Cmd.aEventTransitionText[3]		:= txtEvent_Normal;
Cmd.bEventDetectionEnable		:= FALSE;
Cmd.eEnPlantLock				:= E_BA_LockPriority.eNoLock;
Cmd.eMappingMode				:= E_BA_ByteMappingMode.eBinaryDecimal;
Cmd.eFeedbackMappingMode		:= E_BA_ByteMappingMode.eBinaryDecimal;
END_METHOD

END_FUNCTION_BLOCK

// ---- Templates/POUs/Universal/Control/Monitoring/FB_BA_FdbBinary.TcPOU
{region '#Template'}
	{attribute 'Version' := '5.0.0.0'}
	{attribute 'Tags' := '"LCID": "1031", "Text": "Universal, Control, Monitoring"'}
	{attribute 'Tags' := '"LCID": "1033", "Text": "Universal, Control, Monitoring"'}
	{attribute 'Using' := '"Type": "Template", "URI": "EC_ID"'}
	{attribute 'Using' := '"Type": "Template", "URI": "BA2_Param"'}
	{attribute 'Description' := '"LCID": "1031", "Text": "Überwachung von Signalen"'}
	{attribute 'Description' := '"LCID": "1033", "Text": "Monitoring signals"'}
{endregion}
FUNCTION_BLOCK FB_BA_FdbBinary EXTENDS FB_BA_View
VAR_INPUT
	bEn						: BOOL;	
	bCommand				: BOOL;	
	bFeedback				: BOOL;		
END_VAR
VAR_OUTPUT
	bDst					: BOOL;
END_VAR
VAR_INPUT CONSTANT
	DelayFeedback			: FB_BA_AV_Op;
	Dst						: FB_BA_BV;			
END_VAR
VAR_INPUT CONSTANT PERSISTENT
	{attribute 'parameterUnit':= 's'}
	nInterruptionDelay : UDINT := 1;
END_VAR
VAR
	FdbCtrl					: FB_BA_FdbCtrlBinary;		
END_VAR

SUPER^(); // FB_BA_View
DelayFeedback(); // FB_BA_AV_Op
FdbCtrl(
    bEn := bEn,
    bActuator := bCommand,
    bSwitch := bFeedback,
    nFdbDelay := TO_UDINT(DelayFeedback.fPresentValue),
    nInterruptionDelay := nInterruptionDelay); // FB_BA_FdbCtrlBinary
Dst(bEnPgm := TRUE, bValPgm := FdbCtrl.bQ); // FB_BA_BV
bDst := Dst.bEvent;

METHOD FB_init : BOOL
VAR_INPUT
	bInitRetains : BOOL; // if TRUE, the retain variables are initialized (warm start / cold start)
	bInCopyCode : BOOL;  // if TRUE, the instance afterwards gets moved into the copy code (online change)
END_VAR
DelayFeedback.iParent				:= THIS^;
DelayFeedback.iLabel				:= LblFun_FeedbackDelay;	 	 
DelayFeedback.eUnit 				:= E_BA_Unit.eTime_Seconds;								 
DelayFeedback.fValueRm 				:= 120;
DelayFeedback.fCOVIncrement			:= BA2_Param.fDefCOVIncrement;		

Dst.iParent							:= THIS^;
Dst.iLabel							:= LblFun_Fault;
Dst.sActiveText 					:= txtEvent_Triggered;
Dst.sInactiveText 					:= txtEvent_Normal;
Dst.bEnManualRm						:= FALSE;	//	Priority  8	
Dst.bValManualRm					:= FALSE;	//	Priority  8
Dst.nEventClassID					:= EC_ID.NC30;
Dst.stTimeDelay.nToNormal			:= 0;
Dst.stTimeDelay.nToAbnormal			:= 0;
Dst.bAlarmValue						:= TRUE;
Dst.aEventTransitionText[1]			:= txtEvent_Triggered;
Dst.aEventTransitionText[2]			:= txtEvent_Error;
Dst.aEventTransitionText[3]			:= txtEvent_Normal;
Dst.bEventDetectionEnable			:= TRUE;
Dst.eEnPlantLock					:= E_BA_LockPriority.eNoLock;
END_METHOD

END_FUNCTION_BLOCK

// ---- Templates/POUs/Universal/Control/Object/FB_BA_AV_Op_Val.TcPOU
{region '#Template'}
	{attribute 'Version' := '5.0.0.0'}
	{attribute 'Tags' := '"LCID": "1031", "Text": "Universal, Object, AV"'}
	{attribute 'Tags' := '"LCID": "1033", "Text": "Universal, Sensor, AV"'}
	{attribute 'Using' := '"Type": "Template", "URI": "EC_ID"'}
	{attribute 'Using' := '"Type": "Template", "URI": "BA2_Param"'}
	{attribute 'Description' := '"LCID": "1031", "Text": "AV"'}
	{attribute 'Description' := '"LCID": "1033", "Text": "AV"'}
{endregion}
FUNCTION_BLOCK FB_BA_AV_Op_Val EXTENDS FB_BA_View
VAR_INPUT
	fIn					: REAL;
END_VAR
VAR_OUTPUT
	fPresentValue				: REAL;
END_VAR
VAR_INPUT CONSTANT
	Val					: FB_BA_AV_Op;		
END_VAR
VAR
END_VAR

SUPER^(); // FB_BA_View
Val(fValuePgm := fIn); // FB_BA_AV_Op
fPresentValue := Val.fPresentValue;

METHOD FB_init : BOOL
VAR_INPUT
	bInitRetains : BOOL; // if TRUE, the retain variables are initialized (warm start / cold start)
	bInCopyCode : BOOL;  // if TRUE, the instance afterwards gets moved into the copy code (online change)
END_VAR
Val.iParent					:= THIS^;
Val.iLabel					:= LblFun_MeasuredValue;
Val.eUnit					:= E_BA_Unit.eTemperature_DegreesCelsius;  
Val.fCOVIncrement			:= BA2_Param.fDefCOVIncrement;
END_METHOD

END_FUNCTION_BLOCK

// ---- Templates/POUs/Universal/Control/PID/FB_BA_PID.TcPOU
{region '#Template'}
	{attribute 'Version' := '5.0.0.0'}
	{attribute 'Tags' := '"LCID": "1031", "Text": "Universal, Control, PID, Loop"'}
	{attribute 'Tags' := '"LCID": "1033", "Text": "Universal, Control, PID, Loop"'}
	{attribute 'Using' := '"Type": "Template", "URI": "BA2_Param"'}
	{attribute 'Description' := '"LCID": "1031", "Text": "Regler"'}
	{attribute 'Description' := '"LCID": "1033", "Text": "Controller"'}
{endregion}
FUNCTION_BLOCK FB_BA_PID EXTENDS FB_BA_View
VAR_INPUT
	bEn						: BOOL;
	fW						: REAL;
	fX						: REAL;
	bSync					: BOOL;
	fSync					: REAL;
END_VAR
VAR_OUTPUT
	fY						: REAL;
	fMax					: REAL;
	fMin					: REAL;	
END_VAR
VAR_INPUT CONSTANT		 
	Ctrl					: FB_BA_Loop;	
END_VAR

SUPER^(); // FB_BA_View
Ctrl(bEn := bEn, fSetpoint := fW, fCtrlVal := fX, bEnSync := bSync, fValSync := fSync); // FB_BA_Loop
fY := Ctrl.fPresentValue;
fMin := Ctrl.fMinOutputRm;
fMax := Ctrl.fMaxOutputRm;

METHOD FB_init : BOOL
VAR_INPUT
	bInitRetains : BOOL; // if TRUE, the retain variables are initialized (warm start / cold start)
	bInCopyCode : BOOL;  // if TRUE, the instance afterwards gets moved into the copy code (online change)
END_VAR
Ctrl.iParent				:= THIS^;
Ctrl.iLabel					:= LblFun_LoopObject;   
Ctrl.eOpMode				:= E_BA_PIDMode.ePID;									 	 										 
Ctrl.eOutputUnit			:= E_BA_Unit.eOther_Percent;
Ctrl.eActionRm				:= E_BA_Action.eReverse;
Ctrl.fProportionalConstant	:= 3;
Ctrl.fIntegralConstant		:= 180;
Ctrl.fDerivativeConstant	:= 0;
Ctrl.fMaxOutputRm 			:= 100;
Ctrl.fMinOutputRm			:= 0;
Ctrl.fCOVIncrement			:= 0;
Ctrl.nDampConstant			:= 0;
Ctrl.fNeutralZone			:= 0;
END_METHOD

END_FUNCTION_BLOCK

// ---- Templates/POUs/Universal/Control/Ramp/FB_BA_RampLimitIncrease.TcPOU
{region '#Template'}
	{attribute 'Version' := '5.0.0.0'}
	{attribute 'Tags' := '"LCID": "1031", "Text": "Universal, Control, Ramp limit"'}
	{attribute 'Tags' := '"LCID": "1033", "Text": "Universal, Control, Ramp limit"'}
	{attribute 'Using' := '"Type": "Template", "URI": "BA2_Param"'}
	{attribute 'Description' := '"LCID": "1031", "Text": "Aufsteigende Rampenbegrenzung"'}
	{attribute 'Description' := '"LCID": "1033", "Text": "Rising ramp limit"'}
{endregion}
FUNCTION_BLOCK FB_BA_RampLimitIncrease EXTENDS FB_BA_View 
VAR_INPUT
	bEn			: BOOL;
	bTrig		: BOOL;
END_VAR
VAR_OUTPUT
	fY			: REAL;
END_VAR
VAR_INPUT CONSTANT
	TiUp		: FB_BA_AV_Op;		 										 
	Y			: FB_BA_AV_Op;	
END_VAR
VAR	
	RampFnct	: FB_BA_RampLmt;
	rtrigSync	: R_TRIG;
END_VAR

SUPER^(); // FB_BA_View
TiUp(); // FB_BA_AV_Op
rtrigSync(CLK := bTrig); // R_TRIG
RampFnct(
    bEn := bEn,
    fIn := 100,
    bSync := rtrigSync.Q,
    fSync := 0,
    fHi := 100,
    fLo := 0,
    nTiUp := TO_UDINT(TiUp.fPresentValue),
    nTiDwn := 0); // FB_BA_RampLmt
Y(fValuePgm := RampFnct.fOut); // FB_BA_AV_Op
fY := Y.fPresentValue;

METHOD FB_init : BOOL
VAR_INPUT
	bInitRetains : BOOL; // if TRUE, the retain variables are initialized (warm start / cold start)
	bInCopyCode : BOOL;  // if TRUE, the instance afterwards gets moved into the copy code (online change)
END_VAR
TiUp.iParent				:= THIS^;
TiUp.iLabel					:= LblCtl_RampTimeUp; 	
TiUp.eUnit					:= E_BA_Unit.eTime_Seconds;								 	 
TiUp.fValueRm				:= 600;
TiUp.fCOVIncrement			:= BA2_Param.fDefCOVIncrement;		

	 										 
Y.iParent					:= THIS^;
Y.iLabel					:= LblFun_ControlSignal; 	 	 						 	 
Y.eUnit						:= E_BA_Unit.eOther_Percent;	
Y.fCOVIncrement				:= BA2_Param.fDefCOVIncrement;
END_METHOD

END_FUNCTION_BLOCK

// ---- Templates/POUs/Universal/Control/Scale/FB_BA_Scale_04_Y2_3.TcPOU
{region '#Template'}
	{attribute 'Version' := '5.0.1.0'}
	{attribute 'Tags' := '"LCID": "1031", "Text": "Universal, Control, Scaling"'}
	{attribute 'Tags' := '"LCID": "1033", "Text": "Universal, Control, Scaling"'}
	{attribute 'Using' := '"Type": "Template", "URI": "BA2_Param"'}
	{attribute 'Description' := '"LCID": "1031", "Text": "Skalierung"'}
	{attribute 'Description' := '"LCID": "1033", "Text": "Scaling"'}
{endregion}
FUNCTION_BLOCK FB_BA_Scale_04_Y2_3 EXTENDS FB_BA_View
VAR_INPUT
	fTWth		: REAL;	
END_VAR
VAR_OUTPUT
	fY			: REAL;
END_VAR
VAR_INPUT CONSTANT
	X1			: FB_BA_AV_Op;	
	X2			: FB_BA_AV_Op;	
	X3			: FB_BA_AV_Op;	
	X4			: FB_BA_AV_Op;	
	Y1			: FB_BA_AV_Op;	
	Y2_3		: FB_BA_AV_Op;
	Y4			: FB_BA_AV_Op;
	Y			: FB_BA_AV_Op;				
END_VAR
VAR
	Scale		: FB_BA_Chrct04;	
END_VAR

SUPER^(); // FB_BA_View
X1(); // FB_BA_AV_Op
X2(); // FB_BA_AV_Op
X3(); // FB_BA_AV_Op
X4(); // FB_BA_AV_Op
Y1(); // FB_BA_AV_Op
Y2_3(); // FB_BA_AV_Op
Y4(); // FB_BA_AV_Op
Scale(
    fX := fTWth,
    fX01 := X1.fPresentValue,
    fX02 := X2.fPresentValue,
    fX03 := X3.fPresentValue,
    fX04 := X4.fPresentValue,
    fY01 := Y1.fPresentValue,
    fY02 := Y2_3.fPresentValue,
    fY03 := Y2_3.fPresentValue,
    fY04 := Y4.fPresentValue,
    fYMin := Y2_3.fPresentValue,
    fYMax := Y4.fPresentValue); // FB_BA_Chrct04
Y(fValuePgm := Scale.fCalcVal); // FB_BA_AV_Op
fY := Y.fPresentValue;

METHOD FB_init : BOOL
VAR_INPUT
	bInitRetains : BOOL; // if TRUE, the retain variables are initialized (warm start / cold start)
	bInCopyCode : BOOL;  // if TRUE, the instance afterwards gets moved into the copy code (online change)
END_VAR
X1.iParent			:= THIS^;
X1.iLabel			:= LblCtl_X01;  
X1.sObjectName		:= '{Idx=01}';  						 	 								 	 
X1.eUnit			:= E_BA_Unit.eTemperature_DegreesCelsius;						 	 
X1.fValueRm			:= -15.0;
X1.fCOVIncrement	:= BA2_Param.fDefCOVIncrement;		

X2.iParent			:= THIS^;
X2.iLabel			:= LblCtl_X02;  							 	 
X2.sObjectName		:= '{Idx=02}';  						 	 								 	 
X2.eUnit			:= E_BA_Unit.eTemperature_DegreesCelsius;						 	 
X2.fValueRm			:= -5.0;
X2.fCOVIncrement	:= BA2_Param.fDefCOVIncrement;		

X3.iParent			:= THIS^;
X3.iLabel			:= LblCtl_X03;  						 	 
X3.sObjectName		:= '{Idx=03}';  						 	 								 	 
X3.eUnit			:= E_BA_Unit.eTemperature_DegreesCelsius;						 	 
X3.fValueRm			:= 26.0;
X3.fCOVIncrement	:= BA2_Param.fDefCOVIncrement;		

X4.iParent			:= THIS^;
X4.iLabel			:= LblCtl_X04;  							 	 
X4.sObjectName		:= '{Idx=04}';  						 	 								 	 
X4.eUnit			:= E_BA_Unit.eTemperature_DegreesCelsius;						 	 
X4.fValueRm			:= 32.0;
X4.fCOVIncrement	:= BA2_Param.fDefCOVIncrement;		

Y1.iParent			:= THIS^;
Y1.iLabel			:= LblCtl_Y01;  	
Y1.sObjectName		:= '{Idx=01}';  						 	 								 	 								 	 
Y1.eUnit			:= E_BA_Unit.eTemperature_DegreesCelsius;						 	 
Y1.fValueRm			:= 23.0;
Y1.fCOVIncrement	:= BA2_Param.fDefCOVIncrement;		

Y2_3.iParent		:= THIS^;
Y2_3.iLabel			:= LblCtl_Y02_03;  			
Y2_3.sObjectName	:= '{Idx=02}';  						 	 								 	 								 	 
Y2_3.eUnit			:= E_BA_Unit.eTemperature_DegreesCelsius;						 	 
Y2_3.fValueRm		:= 21.0;
Y2_3.fCOVIncrement	:= BA2_Param.fDefCOVIncrement;		

Y4.iParent			:= THIS^; 
Y4.iLabel			:= LblCtl_Y04; 									 	 
Y4.sObjectName		:= '{Idx=04}';  						 	 								 	 								 	 
Y4.eUnit			:= E_BA_Unit.eTemperature_DegreesCelsius;						 	 
Y4.fValueRm			:= 28.0;
Y4.fCOVIncrement	:= BA2_Param.fDefCOVIncrement;		

Y.iParent			:= THIS^;
Y.iLabel			:= LblFun_SetpointCalculated;		
Y.sObjectName		:= '{Idx=01}';  								 	 
Y.eUnit				:= E_BA_Unit.eTemperature_DegreesCelsius;	
Y.fCOVIncrement		:= BA2_Param.fDefCOVIncrement;
END_METHOD

END_FUNCTION_BLOCK

// ---- Templates/POUs/Universal/Damper/2P/FB_BA_Dmp2P.TcPOU
{region '#Template'}
	{attribute 'Version' := '5.0.0.0'}
	{attribute 'Tags' := '"LCID": "1031", "Text": "Universal, Damper, Aggregate"'}
	{attribute 'Tags' := '"LCID": "1033", "Text": "Universal, Damper, Aggregate"'}
	{attribute 'Using' := '"Type": "Template", "URI": "EC_ID"'}
	{attribute 'Using' := '"Type": "Template", "URI": "BA2_Param"'}
	{attribute 'Description' := '"LCID": "1031", "Text": "2 Punkt Klappe mit Endlagenschalter"'}
	{attribute 'Description' := '"LCID": "1033", "Text": "2 point damper with limit switch"'}
{endregion}			 
FUNCTION_BLOCK FB_BA_Dmp2P EXTENDS FB_BA_ActuatorCmd
VAR_INPUT
END_VAR
VAR_OUTPUT
	bSwiOpn					: BOOL;
	bSwiCls					: BOOL;
END_VAR
VAR_INPUT CONSTANT
	SwiOpn					: FB_BA_BI_Raw;
	SwiCls					: FB_BA_BI_Raw;
	MonitOpen				: FB_BA_FdbBinary;
	MonitClose				: FB_BA_FdbBinary;
END_VAR	
VAR	
END_VAR

SwiOpn(); // FB_BA_BI_Raw
bSwiOpn := SwiOpn.bPresentValue;
SwiCls(); // FB_BA_BI_Raw
bSwiCls := SwiCls.bPresentValue;
SUPER^(); // FB_BA_ActuatorCmd
MonitOpen(bEn := BA2_Param.bDlyStartPLC, bCommand := bCmd, bFeedback := bSwiOpn); // FB_BA_FdbBinary
MonitClose(bEn := BA2_Param.bDlyStartPLC, bCommand := NOT bCmd, bFeedback := bSwiCls); // FB_BA_FdbBinary

METHOD FB_init : BOOL
VAR_INPUT
	bInitRetains : BOOL; // if TRUE, the retain variables are initialized (warm start / cold start)
	bInCopyCode : BOOL;  // if TRUE, the instance afterwards gets moved into the copy code (online change)
END_VAR
SwiOpn.iParent							:= THIS^;
SwiOpn.iLabel							:= LblFun_FeedbackOPEN;  
SwiOpn.sObjectName						:='{Idx=01}';
SwiOpn.ePolarity						:= E_BA_Polarity.eReverse;
SwiOpn.sActiveText 						:= txtEvent_Reached;
SwiOpn.sInactiveText 					:= txtEvent_NotReached;
SwiOpn.nEventClassID					:= EC_ID.NC80;
SwiOpn.stTimeDelay.nToNormal			:= BA2_Param.nDefTimeDelay_ToNormal;
SwiOpn.stTimeDelay.nToAbnormal			:= BA2_Param.nDefTimeDelay_ToAbnormal;
SwiOpn.bAlarmValue						:= TRUE;
SwiOpn.aEventTransitionText[1]			:= txtEvent_Active;
SwiOpn.aEventTransitionText[2]			:= txtEvent_None;
SwiOpn.aEventTransitionText[3]			:= txtEvent_Normal;
SwiOpn.bEventDetectionEnable			:= FALSE;
SwiOpn.eEnPlantLock						:= E_BA_LockPriority.eNoLock;	

SwiCls.iParent							:= THIS^;
SwiCls.iLabel							:= LblFun_FeedbackCLOSED; 
SwiCls.sObjectName						:='{Idx=01}';
SwiCls.ePolarity						:= E_BA_Polarity.eReverse;
SwiCls.sActiveText 						:= txtEvent_Reached;
SwiCls.sInactiveText 					:= txtEvent_NotReached;
SwiCls.nEventClassID					:= EC_ID.NC80;
SwiCls.stTimeDelay.nToNormal			:= BA2_Param.nDefTimeDelay_ToNormal;
SwiCls.stTimeDelay.nToAbnormal			:= BA2_Param.nDefTimeDelay_ToAbnormal;
SwiCls.bAlarmValue						:= TRUE;
SwiCls.aEventTransitionText[1]			:= txtEvent_Active;
SwiCls.aEventTransitionText[2]			:= txtEvent_None;
SwiCls.aEventTransitionText[3]			:= txtEvent_Normal;
SwiCls.bEventDetectionEnable			:= FALSE;
SwiCls.eEnPlantLock						:= E_BA_LockPriority.eNoLock;

MonitOpen.iParent						:= THIS^;
MonitOpen.iLabel						:= LblCtl_FeedbackMonitoring;  
MonitOpen.sObjectName					:='{Idx=01}';
MonitOpen.eDPADMode						:= E_BA_DPADMode.eIncludeDescription;
MonitOpen.DelayFeedback.fValueRm		:= 180.0;
MonitOpen.DelayFeedback.sObjectName		:='{Idx=01}';
MonitOpen.Dst.bEventDetectionEnable		:= TRUE;
MonitOpen.Dst.eEnPlantLock				:= E_BA_LockPriority.eLocalMedium;

MonitClose.iParent						:= THIS^;
MonitClose.iLabel						:= LblCtl_FeedbackMonitoring;
MonitClose.sObjectName					:='{Idx=02}';
MonitClose.eDPADMode					:= E_BA_DPADMode.eIncludeDescription;
MonitClose.DelayFeedback.fValueRm		:= 180.0;
MonitClose.DelayFeedback.iLabel			:= LblFun_FeedbackDelay;
MonitClose.DelayFeedback.sObjectName	:='{Idx=02}';
MonitClose.Dst.iLabel					:= LblFun_Fault;
MonitClose.Dst.sObjectName				:='{Idx=02}';
MonitClose.Dst.bEventDetectionEnable	:= TRUE;
MonitClose.Dst.eEnPlantLock				:= E_BA_LockPriority.eNoLock;
END_METHOD

END_FUNCTION_BLOCK

// ---- Templates/POUs/Universal/Motor/Control/FB_BA_MotCtl.TcPOU
{region '#Template'}
	{attribute 'Version' := '5.0.0.0'}
	{attribute 'Tags' := '"LCID": "1031", "Text": "Universal, Motor, Aggregate"'}
	{attribute 'Tags' := '"LCID": "1033", "Text": "Universal, Motor, Aggregate"'}
	{attribute 'Using' := '"Type": "Template", "URI": "EC_ID"'}
	{attribute 'Using' := '"Type": "Template", "URI": "BA2_Param"'}
	{attribute 'Description' := '"LCID": "1031", "Text": "Motor modulierend mit Regler"'}
	{attribute 'Description' := '"LCID": "1033", "Text": "Motor modulating with controller"'}
{endregion}		
FUNCTION_BLOCK FB_BA_MotCtl EXTENDS FB_BA_View
VAR_INPUT
	fIn				: REAL;	// Istwert Regler // Actual value controller	
	stCmd			: ST_BA_Mdlt;
END_VAR
VAR_OUTPUT
	bCmd			: BOOL;
	fMdlt			: REAL;
	bDst			: BOOL;
	eActivePrio		: E_BA_Priority;
END_VAR

VAR_INPUT CONSTANT
	Dst				: FB_BA_BI_Raw;
	Cmd				: FB_BA_BO_Raw;								 
	Mdlt			: FB_BA_AO_Raw;							
	Sp				: FB_BA_AV_Op;		 
	Ctrl			: FB_BA_Loop;		
	PlantLock		: FB_BA_PlantLock;														
END_VAR
VAR
	bPrioSfty					: BOOL;
	bPrioCrit					: BOOL;	
	
	PrioSwiVal					: FB_BA_PrioSwi_UDI04;	

	MuxCmd						: FB_BA_MMUX_B04;
	MuxMdlt						: FB_BA_MMUX_R04;
	fMax						: REAL;
	fMin						: REAL;		
END_VAR
VAR // added by the converter: edge detectors and wires of the graphical bodies
    _w1, _w2 : ANY;
END_VAR

SUPER^(); // FB_BA_View
Dst(); // FB_BA_BI_Raw
PlantLock(); // FB_BA_PlantLock
bPrioSfty := PlantLock.bPrioHigh OR PlantLock.bPrioLocalHigh;
bPrioCrit := PlantLock.bPrioMedium OR PlantLock.bPrioLocalMedium;
bDst := bPrioSfty OR bPrioCrit;
PrioSwiVal(
    bEn01 := stCmd.bEnSfty,
    nVal01 := stCmd.eValSfty,
    bEn02 := stCmd.bEnCrit,
    nVal02 := stCmd.eValCrit,
    bEn03 := stCmd.bEnPgm,
    nVal03 := stCmd.eValPgm); // FB_BA_PrioSwi_UDI04
MuxCmd(
    bEn := TRUE,
    nSel := PrioSwiVal.nVal,
    nEn01 := E_BA_Mdlt.eOff,
    bVal01 := FALSE,
    nEn02 := E_BA_Mdlt.eOn,
    bVal02 := TRUE,
    nEn03 := E_BA_Mdlt.eMin,
    bVal03 := TRUE,
    nEn04 := E_BA_Mdlt.eMax,
    bVal04 := TRUE); // FB_BA_MMUX_B04
Cmd(
    bEnSfty := stCmd.bEnSfty OR bPrioSfty,
    bValSfty := SEL(bPrioSfty, MuxCmd.bVal, FALSE),
    bEnCrit := stCmd.bEnCrit OR bPrioCrit,
    bValCrit := _w1,
    bEnPgm := stCmd.bEnPgm,
    bValPgm := MuxCmd.bVal); // FB_BA_BO_Raw
_w1 := SEL(bPrioCrit, MuxCmd.bVal, FALSE);
bCmd := Cmd.bPresentValue;
eActivePrio := Cmd.eActivePrio;
Ctrl(bEn := bCmd, fSetpoint := Sp.fPresentValue, fCtrlVal := fIn); // FB_BA_Loop
Sp(); // FB_BA_AV_Op
fMin := Ctrl.fMinOutputRm;
fMax := Ctrl.fMaxOutputRm;
MuxMdlt(
    bEn := bCmd,
    nSel := PrioSwiVal.nVal,
    nEn01 := E_BA_Mdlt.eOff,
    fVal01 := 0,
    nEn02 := E_BA_Mdlt.eOn,
    fVal02 := Ctrl.fPresentValue,
    nEn03 := E_BA_Mdlt.eMin,
    fVal03 := fMin,
    nEn04 := E_BA_Mdlt.eMax,
    fVal04 := fMax); // FB_BA_MMUX_R04
Mdlt(
    bEnSfty := Cmd.bEnSfty,
    fValSfty := SEL(bPrioSfty, MuxMdlt.fVal, 0),
    bEnCrit := Cmd.bEnCrit,
    fValCrit := _w2,
    bEnPgm := Cmd.bEnPgm,
    fValPgm := MuxMdlt.fVal); // FB_BA_AO_Raw
_w2 := SEL(bPrioCrit, MuxMdlt.fVal, 0);
fMdlt := Mdlt.fPresentValue;

METHOD FB_init : BOOL
VAR_INPUT
	bInitRetains : BOOL; // if TRUE, the retain variables are initialized (warm start / cold start)
	bInCopyCode : BOOL;  // if TRUE, the instance afterwards gets moved into the copy code (online change)
END_VAR
PlantLock.Parent					:= THIS^;		

Dst.iParent							:= THIS^;
Dst.iLabel							:= LblFun_Fault;  
Dst.ePolarity						:= E_BA_Polarity.eReverse;
Dst.sActiveText 					:= txtEvent_Triggered;
Dst.sInactiveText 					:= txtEvent_Normal;
Dst.nEventClassID					:= EC_ID.NC30;
Dst.stTimeDelay.nToNormal			:= BA2_Param.nDefTimeDelay_ToNormal;
Dst.stTimeDelay.nToAbnormal			:= BA2_Param.nDefTimeDelay_ToAbnormal;
Dst.bAlarmValue						:= TRUE;
Dst.aEventTransitionText[1]			:= txtEvent_Triggered;
Dst.aEventTransitionText[2]			:= txtEvent_Error;
Dst.aEventTransitionText[3]			:= txtEvent_Normal;
Dst.bEventDetectionEnable			:= TRUE;
Dst.eEnPlantLock					:= E_BA_LockPriority.eLocalMedium;

Cmd.iParent							:= THIS^;
Cmd.iLabel							:= LblFun_SwitchingCommand;  
Cmd.ePolarity						:= E_BA_Polarity.eNormal;
Cmd.sActiveText 					:= txtEvent_On;
Cmd.sInactiveText 					:= txtEvent_Off;
Cmd.bEnManualRm						:= FALSE;	//	Priority  8	
Cmd.bValManualRm					:= FALSE;	//	Priority  8
Cmd.nEventClassID					:= EC_ID.NC40;
Cmd.stTimeDelay.nToNormal			:= BA2_Param.nDefTimeDelay_ToNormal;
Cmd.stTimeDelay.nToAbnormal			:= BA2_Param.nDefTimeDelay_ToAbnormal;
Cmd.aEventTransitionText[1]			:= txtEvent_Disturb;
Cmd.aEventTransitionText[2]			:= txtEvent_None;
Cmd.aEventTransitionText[3]			:= txtEvent_Normal;
Cmd.bEventDetectionEnable			:= FALSE;
Cmd.eEnPlantLock					:= E_BA_LockPriority.eNoLock;

Mdlt.iParent						:= THIS^;
Mdlt.iLabel							:= LblFun_ControlSignal;  
Mdlt.eUnit							:= E_BA_Unit.eOther_Percent;
Mdlt.fResolution 					:= 0.003051851;
Mdlt.fScaleOffset 					:= 0;
Mdlt.fCOVIncrement					:= BA2_Param.fDefCOVIncrement;
Mdlt.bEnManualRm					:= FALSE;	//	Priority  8	
Mdlt.fValManualRm					:= 0.0;		//	Priority  8
Mdlt.nEventClassID					:= EC_ID.NC80;
Mdlt.stTimeDelay.nToNormal			:= BA2_Param.nDefTimeDelay_ToNormal;
Mdlt.stTimeDelay.nToAbnormal		:= BA2_Param.nDefTimeDelay_ToAbnormal;
Mdlt.stHighLimit.bEnable			:= FALSE;
Mdlt.stHighLimit.fValue				:= 0.0;		
Mdlt.stLowLimit.bEnable				:= FALSE;
Mdlt.stLowLimit.fValue				:= 0.0;
Mdlt.fLimitDeadband 				:= BA2_Param.fDefLimitDeadband;
Mdlt.aEventTransitionText[1]		:= txtEvent_Disturb;
Mdlt.aEventTransitionText[2]		:= txtEvent_None;
Mdlt.aEventTransitionText[3]		:= txtEvent_Normal;
Mdlt.bEventDetectionEnable			:= FALSE;
Mdlt.eEnPlantLock					:= E_BA_LockPriority.eNoLock;

Sp.iParent							:= THIS^;
Sp.iLabel							:= LblFun_Setpoint; 
Sp.eUnit 							:= E_BA_Unit.ePressure_Pascals;								 
Sp.fValueRm							:= 250;
Sp.fCOVIncrement					:= BA2_Param.fDefCOVIncrement;

Ctrl.iParent						:= THIS^;
Ctrl.iLabel							:= LblFun_LoopObject;  
Ctrl.eOpMode						:= E_BA_PIDMode.ePID;								 	 										 
Ctrl.eOutputUnit					:= E_BA_Unit.eOther_Percent;
Ctrl.eActionRm						:= E_BA_Action.eReverse;
Ctrl.fProportionalConstant			:= 0.01;
Ctrl.fIntegralConstant				:= 60;
Ctrl.fDerivativeConstant			:= 0;
Ctrl.fMaxOutputRm 					:= 100;
Ctrl.fMinOutputRm					:= 20;
Ctrl.fCOVIncrement					:= 0;
Ctrl.nDampConstant					:= 0;
Ctrl.fNeutralZone					:= 0;
END_METHOD

END_FUNCTION_BLOCK

// ---- Templates/POUs/Universal/Motor/Control/FB_BA_MotCtlExt.TcPOU
{region '#Template'}
	{attribute 'Version' := '5.0.0.0'}
	{attribute 'Tags' := '"LCID": "1031", "Text": "Universal, Motor, Aggregate"'}
	{attribute 'Tags' := '"LCID": "1033", "Text": "Universal, Motor, Aggregate"'}
	{attribute 'Using' := '"Type": "Template", "URI": "EC_ID"'}
	{attribute 'Using' := '"Type": "Template", "URI": "BA2_Param"'}
	{attribute 'Description' := '"LCID": "1031", "Text": "Motor modulierend mit Regler erweitert"'}
	{attribute 'Description' := '"LCID": "1033", "Text": "Motor modulating with controller extended"'}
{endregion}		 
FUNCTION_BLOCK FB_BA_MotCtlExt EXTENDS FB_BA_MotCtl
VAR_INPUT CONSTANT
	ThOvrld			: FB_BA_BI_Raw;							
	MntnSwi			: FB_BA_BI_Raw;
END_VAR
VAR
END_VAR

ThOvrld(); // FB_BA_BI_Raw
MntnSwi(); // FB_BA_BI_Raw
SUPER^(); // FB_BA_MotCtl

METHOD FB_init : BOOL
VAR_INPUT
	bInitRetains : BOOL; // if TRUE, the retain variables are initialized (warm start / cold start)
	bInCopyCode : BOOL;  // if TRUE, the instance afterwards gets moved into the copy code (online change)
END_VAR
ThOvrld.iParent						:= THIS^;
ThOvrld.iLabel						:= LblFun_Fault;  
ThOvrld.ePolarity					:= E_BA_Polarity.eReverse;
ThOvrld.sActiveText 				:= txtEvent_Triggered;
ThOvrld.sInactiveText 				:= txtEvent_Normal;
ThOvrld.nEventClassID				:= EC_ID.NC30;
ThOvrld.stTimeDelay.nToNormal		:= BA2_Param.nDefTimeDelay_ToNormal;
ThOvrld.stTimeDelay.nToAbnormal		:= BA2_Param.nDefTimeDelay_ToAbnormal;
ThOvrld.bAlarmValue					:= TRUE;
ThOvrld.aEventTransitionText[1]		:= txtEvent_Triggered;
ThOvrld.aEventTransitionText[2]		:= txtEvent_Error;
ThOvrld.aEventTransitionText[3]		:= txtEvent_Normal;
ThOvrld.bEventDetectionEnable		:= TRUE;
ThOvrld.eEnPlantLock				:= E_BA_LockPriority.eLocalMedium;	

MntnSwi.iParent						:= THIS^;
MntnSwi.iLabel						:= LblFun_MaintenanceMessage;  
MntnSwi.ePolarity					:= E_BA_Polarity.eReverse;
MntnSwi.sActiveText 				:= txtEvent_Maintenace;
MntnSwi.sInactiveText 				:= txtEvent_Normal;
MntnSwi.nEventClassID				:= EC_ID.NC50;
MntnSwi.stTimeDelay.nToNormal		:= BA2_Param.nDefTimeDelay_ToNormal;
MntnSwi.stTimeDelay.nToAbnormal		:= BA2_Param.nDefTimeDelay_ToAbnormal;
MntnSwi.bAlarmValue					:= TRUE;
MntnSwi.aEventTransitionText[1]		:= txtEvent_Disturb;
MntnSwi.aEventTransitionText[2]		:= txtEvent_None;
MntnSwi.aEventTransitionText[3]		:= txtEvent_Normal;
MntnSwi.bEventDetectionEnable		:= TRUE;
MntnSwi.eEnPlantLock				:= E_BA_LockPriority.eLocalMedium;
END_METHOD

END_FUNCTION_BLOCK

// ---- Templates/POUs/Universal/WeatherStation/Thies/FB_BA_ThiesData.TcPOU
{region '#Template'}
	{attribute 'Version' := '5.1.1.0'}
	{attribute 'Tags' := '"LCID": "1031", "Text": "Universal, Weather station, Thies"'}
	{attribute 'Tags' := '"LCID": "1033", "Text": "Universal, Weather station, Thies"'}
	{attribute 'Using' := '"Type": "Template", "URI": "ST_BA_WSC11Data"'}		 
	{attribute 'Using' := '"Type": "Template", "URI": "ST_BA_WSC11Status"'}
	{attribute 'Using' := '"Type": "Template", "URI": "ST_BA_WeatherStation"'}
	{attribute 'Description' := '"LCID": "1031", "Text": "Rangierverteiler der gewünschen Daten"'}
	{attribute 'Description' := '"LCID": "1033", "Text": "Data collector of important data"'}
{endregion}
FUNCTION_BLOCK FB_BA_ThiesData
VAR_INPUT
	stWSC11Data				: ST_BA_WSC11Data;
	bHold					: BOOL;
END_VAR
VAR
	_stWeatherStation		: ST_BA_WeatherStation;
END_VAR
VAR_OUTPUT
	stWeatherStation		: ST_BA_WeatherStation;
END_VAR



	stWeatherStation.fLatitude				:=	stWSC11Data.fLatitude;
	stWeatherStation.fLongitude				:=	stWSC11Data.fLongitude;			
	stWeatherStation.fSunAzimuth			:=	stWSC11Data.fSunAzimuth;			
	stWeatherStation.fSunElevation			:=	stWSC11Data.fSunElevation;
	stWeatherStation.bRain					:=	stWSC11Data.bRain;
	stWeatherStation.stDateTime				:=	stWSC11Data.stDateTime;
	stWeatherStation.fOutsideTemperature	:=	stWSC11Data.fOutsideTemperature;	
	stWeatherStation.fDewPointTemperature	:=	stWSC11Data.fDewPointTemperature;
	stWeatherStation.fPressureAbs			:=	stWSC11Data.fPressureAbs;	
	stWeatherStation.fPressureRel			:=	stWSC11Data.fPressureRel;	
	stWeatherStation.fHumidityAbs			:=	stWSC11Data.fHumidityAbs;	
	stWeatherStation.fHumidityRel			:=	stWSC11Data.fHumidityRel;
	stWeatherStation.fBrightnessEast		:=	stWSC11Data.fBrightnessEast * 1000;			
	stWeatherStation.fBrightnessNorth		:=	stWSC11Data.fBrightnessNorth * 1000;
	stWeatherStation.fBrightnessSouth		:=	stWSC11Data.fBrightnessSouth * 1000;	
	stWeatherStation.fBrightnessWest		:=	stWSC11Data.fBrightnessWest * 1000;
	stWeatherStation.fDawn					:=	stWSC11Data.fDawn;	
	stWeatherStation.fGlobalRadiation		:=	stWSC11Data.fGlobalRadiation;
	stWeatherStation.fWindDirection			:=	stWSC11Data.fWindDirection;			
	stWeatherStation.fWindSpeed				:=	stWSC11Data.fWindSpeed;	
	
	IF bHold	THEN
		stWeatherStation					:= _stWeatherStation;
	END_IF
	
	_stWeatherStation						:= stWeatherStation;

END_FUNCTION_BLOCK

// ---- Templates/POUs/Universal/WeatherStation/Thies/FB_BA_ThiesWSC11.TcPOU
{region '#Template'}
	{attribute 'Version' := '5.0.0.0'}
	{attribute 'Tags' := '"LCID": "1031", "Text": "Universal, Weather station, Thies"'}
	{attribute 'Tags' := '"LCID": "1033", "Text": "Universal, Weather station, Thies"'}
	{attribute 'Using' := '"Type": "Template", "URI": "ST_BA_WSC11Data"'}		 
	{attribute 'Using' := '"Type": "Template", "URI": "ST_BA_WSC11Status"'}
	{attribute 'Description' := '"LCID": "1031", "Text": "Konfguration der Wetterstation und Auswerten des Telegramms"'}
	{attribute 'Description' := '"LCID": "1033", "Text": "Configuration of the weatherstation and extracting the data out of the telegram"'}
{endregion}
FUNCTION_BLOCK FB_BA_ThiesWSC11
VAR_INPUT
	bRst					: BOOL;				// reset weather-station
END_VAR                                     	
VAR_INPUT CONSTANT PERSISTENT               	
	{attribute 'parameterUnit':= 'ms'}      	
	nUpdateTime				: UDINT := 500;		// data-polling interval [500..60000ms]
	{attribute 'parameterUnit':= 's'}      	
	nConfigTimeout			: UDINT	:= 10;		// Timeout for configutation-routine
	{attribute 'parameterUnit':= ''}        	
	nMaxCyclesOldData		: UDINT	:= 5;		// No change of data: counting polling-cycles with identical data before sending an error; min=2
	{attribute 'parameterUnit':= 'min'}     	
	nWndDatAvrgIntVal		: UDINT;			// Wind data averaging intervall - 0 = Off; 1-10 = minutes
	bWndSpdLEDOn			: BOOL;				// Wind speed LED on - FALSE = blue LED Off ; TRUE = blue LED On
	bTwiLgtCalcAvrg			: BOOL;				// Twilight-caluclation average - FALSE = Sum of the light-sensors is taken ; TRUE = Average of the light-sensors is taken
	{attribute 'parameterUnit':= 'deg'} 		
	nWndDirNorthOffs		: UDINT;			// Wind direction North offset (correction) [0..360°]
	{attribute 'parameterUnit':= 'm'}   		
	nStHgtAMSL				: UDINT;			// Station height above mean sea level [0..3000m], 3001 means, that the level is automatically taken from GPS-device			
	{attribute 'parameterUnit':= 's'}							
	nRainOffDly				: UDINT;			// Rain off delay [0..3600s]					
	{attribute 'parameterUnit':= 's'}							
	nDistMsgDly				: UDINT;			// Disturbance message delay [0..60s]
END_VAR
VAR_OUTPUT
	stWSC11Data				: ST_BA_WSC11Data;
	bErr					: BOOL;				// error
	sErrDescr				: T_MaxString;		// error description
END_VAR                     
VAR_IN_OUT                  
	TXBuffer				: ComBuffer;
	RXBuffer				: ComBuffer;
END_VAR                     
VAR                
	tUpdateTime				: TIME;
	tRainOffDly				: TIME;
	tDistMsgDly				: TIME;
	                        
	rtRst					: R_TRIG;
	tonTimeout				: TON;
	tonSendParam			: TON;
	tonReadData				: TON;
	tofRain					: TOF;
	tonDist					: ARRAY[1..21]OF TON;
	SendString				: SendString;
	ReceiveString			: ReceiveString;
	ReceiveStringMValues	: ReceiveString255;
	bOldData				: BOOL;					// no data change for "nMaxCyclesOldData" polling-cycles
	bThiesConfigError		: BOOL;					// timeout-error configurating the Thies-weather-station
                            
	nStep					: INT;
	nLastStep				: INT;
	bSendParameter			: BOOL;
	bFeedbackParameter		: BOOL;
	sReceivedParameter		: STRING;
                            
	sMValues				: STRING(255);
	sMValues_LC				: STRING(255);
	nPollingCounter			: UDINT;
                            
	sDateAndTime			: STRING;
	sStatus					: STRING;
	dwStatus				: DWORD;
                            
	nWndDatAvrgIntVal_Mem	: UDINT;
	bWndSpdLEDOn_Mem		: BOOL;
	bTwiLgtCalcAvrg_Mem		: BOOL;
	nWndDirNorthOffs_Mem	: UDINT;
	nStHgtAMSL_Mem			: UDINT;
                            
	sWndDatAvrgIntVal		: STRING;
	sWndDirNorthOffs		: STRING;
	sStHgtAMSL				: STRING;			// Height Above Mean Sea Level
END_VAR


// limiting of input-values
nUpdateTime			:= LIMIT (500, nUpdateTime, 60000);
nMaxCyclesOldData	:= MAX (2, nMaxCyclesOldData);
nWndDatAvrgIntVal 	:= LIMIT (0, nWndDatAvrgIntVal, 10);
nWndDirNorthOffs	:= LIMIT (0, nWndDirNorthOffs, 360);
nStHgtAMSL			:= LIMIT (0, nStHgtAMSL, 3001);
nRainOffDly			:= LIMIT (0, nRainOffDly, 3600);
nDistMsgDly			:= LIMIT (0, nDistMsgDly, 60);

tUpdateTime			:= TO_TIME(nUpdateTime);
tRainOffDly			:= TO_TIME(nRainOffDly*1000);
tDistMsgDly			:= TO_TIME(nDistMsgDly*1000);

// watch for input-changes
rtRst(CLK:=bRst );

IF rtRst.Q
OR nWndDatAvrgIntVal		<> nWndDatAvrgIntVal_Mem
OR bWndSpdLEDOn				<> bWndSpdLEDOn_Mem
OR bTwiLgtCalcAvrg			<> bTwiLgtCalcAvrg_Mem
OR nWndDirNorthOffs			<> nWndDirNorthOffs_Mem
OR nStHgtAMSL				<> nStHgtAMSL_Mem		 THEN                     
  
	bWndSpdLEDOn_Mem		:= bWndSpdLEDOn;
	bTwiLgtCalcAvrg_Mem		:= bTwiLgtCalcAvrg;
	nWndDirNorthOffs_Mem	:= nWndDirNorthOffs;
	nStHgtAMSL_Mem			:= nStHgtAMSL;
	nWndDatAvrgIntVal_Mem	:= nWndDatAvrgIntVal;
	
	bSendParameter			:= TRUE;       
	nStep					:= 0;
END_IF

tonTimeout(IN:=bSendParameter, PT:= F_BA_UdiToTiSec(nConfigTimeout));
IF tonTimeout.Q	THEN
	bThiesConfigError	:= TRUE;
	tonTimeout			(IN:= FALSE);
	nStep				:= 0;		// restart
END_IF

CASE nStep OF

// sequence: send changed parameters
	0:
		tonSendParam(IN:=bSendParameter , PT:=tUpdateTime+T#1S);
			IF tonSendParam.Q AND bSendParameter THEN
				nStep:=2;
			END_IF

	1:
		ReceiveString(
					Prefix:= ,
					Suffix:='$0D',
					ReceivedString:=sReceivedParameter,
					RXbuffer:=RXBuffer);
		IF ReceiveString.StringReceived THEN
			bFeedbackParameter:=TRUE;
		END_IF
		IF NOT ReceiveString.Busy AND bFeedbackParameter THEN
			bFeedbackParameter:=FALSE;
			nStep:=nLastStep+1;
		END_IF

	2:	// set password
		SendString(
				SendString:='00KY234$0D' ,
				TXbuffer:=TXBuffer );
		nLastStep:=2;
		nStep:=1;

	3:	// Wind data averaging interval
		sWndDatAvrgIntVal:='00AI';
		sWndDatAvrgIntVal:=CONCAT(sWndDatAvrgIntVal,TO_STRING(nWndDatAvrgIntVal_Mem));
		sWndDatAvrgIntVal:=CONCAT(sWndDatAvrgIntVal,'$0D');
		SendString(
				SendString:=sWndDatAvrgIntVal ,
				TXbuffer:=TXBuffer );
		nLastStep:=3;
		nStep:=1;

	4:	// Wind speed LED
		IF bWndSpdLEDOn THEN
		SendString(
				SendString:='00LC0$0D' ,
				TXbuffer:=TXBuffer );
		ELSE
		SendString(
				SendString:='00LC1$0D' ,
				TXbuffer:=TXBuffer );
		END_IF
		nLastStep:=4;
		nStep:=1;

	5:	// Twilight-caluclation
		IF bTwiLgtCalcAvrg THEN
		SendString(
				SendString:='00DC1$0D' ,
				TXbuffer:=TXBuffer );
		ELSE
		SendString(
				SendString:='00DC0$0D' ,
				TXbuffer:=TXBuffer );
		END_IF
		nLastStep:=5;
		nStep:=1;

	6:	// Wind direction North offset
		sWndDirNorthOffs:='00DO';
		sWndDirNorthOffs:=CONCAT(sWndDirNorthOffs,TO_STRING(nWndDirNorthOffs));
		sWndDirNorthOffs:=CONCAT(sWndDirNorthOffs,'$0D');
		SendString(
				SendString:=sWndDirNorthOffs ,
				TXbuffer:=TXBuffer );
		nLastStep:=6;
		nStep:=1;

	7:	// Station height above mean seal level
		sStHgtAMSL:='00SH';
		sStHgtAMSL:=CONCAT(sStHgtAMSL,TO_STRING(nStHgtAMSL));
		sStHgtAMSL:=CONCAT(sStHgtAMSL,'$0D');
		SendString(
				SendString:=sStHgtAMSL ,
				TXbuffer:=TXBuffer );
		nLastStep:=7;
		nStep:=1;

	8:	// Reset
		IF bRst THEN
		SendString(
				SendString:='00RS02$0D' ,
				TXbuffer:=TXBuffer );
		nLastStep:=8;
		nStep:=1;
		ELSE
		nStep:=9;
		END_IF

	9:
		bSendParameter		:= FALSE;
		bThiesConfigError	:= FALSE;
		nLastStep			:= 9;
		nStep				:= 0;

END_CASE

// read data periodically
sMValues_LC	:= sMValues;	// Last cycle -> detect changes

tonReadData(IN:=NOT tonReadData.Q AND NOT bSendParameter , PT:=tUpdateTime);

IF tonReadData.Q THEN
	nPollingCounter	:= nPollingCounter+1;
	SendString(
	SendString:='00TR1$0D' ,
	TXbuffer:=TXBuffer );
END_IF

ReceiveStringMValues(
	Prefix:='$02WSC' ,
	Suffix:='$0D$0A' ,
	Timeout:=T#3s ,
	ReceivedString:=sMValues ,
	RXbuffer:=RXBuffer);
	
IF (sMValues_LC	= sMValues)	THEN
	IF nPollingCounter > nMaxCyclesOldData	THEN
		nPollingCounter := nMaxCyclesOldData;
		bOldData		:= TRUE;
	END_IF
ELSE
	bOldData		:= FALSE;
	nPollingCounter	:= 0;
END_IF

IF ReceiveStringMValues.StringReceived THEN
	
	// date and time from weather-station
	
	sDateAndTime:='DT#';
	sDateAndTime:=CONCAT(sDateAndTime,MID(sMValues,4,15));
	sDateAndTime:=CONCAT(sDateAndTime,'-');
	sDateAndTime:=CONCAT(sDateAndTime,MID(sMValues,2,12));
	sDateAndTime:=CONCAT(sDateAndTime,'-');
	sDateAndTime:=CONCAT(sDateAndTime,MID(sMValues,2,9));
	sDateAndTime:=CONCAT(sDateAndTime,'-');
	sDateAndTime:=CONCAT(sDateAndTime,MID(sMValues,2,20));
	sDateAndTime:=CONCAT(sDateAndTime,':');
	sDateAndTime:=CONCAT(sDateAndTime,MID(sMValues,2,23));
	sDateAndTime:=CONCAT(sDateAndTime,':');
	sDateAndTime:=CONCAT(sDateAndTime,MID(sMValues,2,26));
	
	stWSC11Data.stDateTime				:= DT_TO_SYSTEMTIME(TO_DT(sDateAndTime));
										
	stWSC11Data.sTimeFormat				:= MID(sMValues,6,29);
										
	
	// weather-data from weather-station
	
	stWSC11Data.fBrightnessNorth		:= TO_REAL(MID(sMValues,5,36));
	stWSC11Data.fBrightnessEast			:= TO_REAL(MID(sMValues,5,42));
	stWSC11Data.fBrightnessSouth		:= TO_REAL(MID(sMValues,5,48));
	stWSC11Data.fBrightnessWest			:= TO_REAL(MID(sMValues,5,54));
										   
	stWSC11Data.fDawn					:= TO_REAL(STRING_TO_INT(MID(sMValues,3,60)));
										   
	stWSC11Data.fGlobalRadiation		:= TO_INT(MID(sMValues,4,64));
										   
	stWSC11Data.fOutsideTemperature		:= TO_REAL(MID(sMValues,5,69));
										   
	tofRain								(IN	:= TO_BOOL(TO_BYTE(MID(sMValues,1,75))) , PT:=tRainOffDly);
	stWSC11Data.bRain					:= tofRain.Q;
										   
	stWSC11Data.fWindSpeed				:= TO_REAL(MID(sMValues,4,77));
	stWSC11Data.fWindDirection			:= TO_REAL(TO_INT(MID(sMValues,3,82)));
										   
	stWSC11Data.fPressureAbs			:= TO_REAL(MID(sMValues,6,86));
	stWSC11Data.fPressureRel			:= TO_REAL(MID(sMValues,6,93));
										   
	stWSC11Data.fCaseTemperature		:= TO_REAL(MID(sMValues,5,100));
										   
	stWSC11Data.fHumidityRel			:= TO_REAL(MID(sMValues,5,106));
	stWSC11Data.fHumidityAbs			:= TO_REAL(MID(sMValues,6,112));
										   
	stWSC11Data.fDewPointTemperature	:= TO_REAL(MID(sMValues,5,119));
										   
	stWSC11Data.fLongitude				:= TO_REAL(TO_LREAL(MID(sMValues,11,125)));
	stWSC11Data.fLatitude				:= TO_REAL(TO_LREAL(MID(sMValues,10,137)));
										   
	stWSC11Data.fSunElevation			:= TO_REAL(MID(sMValues,5,148));
	stWSC11Data.fSunAzimuth				:= TO_REAL(MID(sMValues,5,154));
	
	
	// status of the weather-station
	
	sStatus:=MID(sMValues,2,166);
	sStatus:=CONCAT(sStatus,MID(sMValues,2,164));
	sStatus:=CONCAT(sStatus,MID(sMValues,2,162));
	sStatus:=CONCAT(sStatus,MID(sMValues,2,160));
	
	HEXSTR_TO_DATA(sStatus, ADR(dwStatus), 4);
	
	tonDist[01](IN:=dwStatus.00 , PT:=tDistMsgDly , Q=>stWSC11Data.stStatus.bDewProtection );
	tonDist[02](IN:=dwStatus.01 , PT:=tDistMsgDly , Q=>stWSC11Data.stStatus.bSensorDryingPeriod );
	tonDist[03](IN:=dwStatus.02 , PT:=tDistMsgDly , Q=>stWSC11Data.stStatus.bInvalidRMC_Telegramm );
	tonDist[04](IN:=dwStatus.03 , PT:=tDistMsgDly , Q=>stWSC11Data.stStatus.bInvalidGPS_Time );
	tonDist[05](IN:=dwStatus.04 , PT:=tDistMsgDly , Q=>stWSC11Data.stStatus.bInvalidDataAD_Converter );
	tonDist[06](IN:=dwStatus.05 , PT:=tDistMsgDly , Q=>stWSC11Data.stStatus.bInvalidDataPressureSensor );
	tonDist[07](IN:=dwStatus.06 , PT:=tDistMsgDly , Q=>stWSC11Data.stStatus.bInvalidDataBrightnessSensorNorth );
	tonDist[08](IN:=dwStatus.07 , PT:=tDistMsgDly , Q=>stWSC11Data.stStatus.bInvalidDataBrightnessSensorEast );
	tonDist[09](IN:=dwStatus.08 , PT:=tDistMsgDly , Q=>stWSC11Data.stStatus.bInvalidDataBrightnessSensorSouth );
	tonDist[10](IN:=dwStatus.09 , PT:=tDistMsgDly , Q=>stWSC11Data.stStatus.bInvalidDataBrightnessSensorWest );
	tonDist[11](IN:=dwStatus.10 , PT:=tDistMsgDly , Q=>stWSC11Data.stStatus.bInvalidDataTwilightSensor );
	tonDist[12](IN:=dwStatus.11 , PT:=tDistMsgDly , Q=>stWSC11Data.stStatus.bInvalidDataSolarRadiationSensor );
	tonDist[13](IN:=dwStatus.12 , PT:=tDistMsgDly , Q=>stWSC11Data.stStatus.bInvalidDataOutsideTemperatureSensor );
	tonDist[14](IN:=dwStatus.13 , PT:=tDistMsgDly , Q=>stWSC11Data.stStatus.bInvalidDataRainSensor );
	tonDist[15](IN:=dwStatus.14 , PT:=tDistMsgDly , Q=>stWSC11Data.stStatus.bInvalidDataWindSpeedSensor );
	tonDist[16](IN:=dwStatus.15 , PT:=tDistMsgDly , Q=>stWSC11Data.stStatus.bInvalidDataWindDirectionSensor );
	tonDist[17](IN:=dwStatus.16 , PT:=tDistMsgDly , Q=>stWSC11Data.stStatus.bInvalidDataHumiditySensor );
	tonDist[18](IN:=dwStatus.17 , PT:=tDistMsgDly , Q=>stWSC11Data.stStatus.bLatestRestartByWatchdogReset );
	tonDist[19](IN:=dwStatus.18 , PT:=tDistMsgDly , Q=>stWSC11Data.stStatus.bInvalidEEPROM_Parameters );
	tonDist[20](IN:=dwStatus.19 , PT:=tDistMsgDly , Q=>stWSC11Data.stStatus.bDefaultEEPROM_Parameters );
	tonDist[21](IN:=dwStatus.20 , PT:=tDistMsgDly , Q=>stWSC11Data.stStatus.bLatestRestartWithNewFirmware );

END_IF

bErr		:= FALSE;
sErrDescr	:= ''; 

IF bOldData	THEN
	bErr		:= TRUE;
	sErrDescr	:= 'Data unchanged for nMaxCyclesOldData (parameter)'; 
END_IF

IF bThiesConfigError	THEN
	bErr		:= TRUE;
	sErrDescr	:= 'Timeout-error while configurating the weather-station'; 
END_IF

END_FUNCTION_BLOCK
